C01799=1100.820,324.418,-83.531,179.191,17.633,151.939
C01800=1100.814,324.171,-83.499,179.188,17.631,151.939
C01801=1100.808,323.923,-83.467,179.185,17.628,151.939
C01802=1100.802,323.675,-83.435,179.182,17.626,151.939
C01803=1100.797,323.427,-83.403,179.179,17.624,151.939
C01804=1100.791,323.179,-83.370,179.175,17.622,151.939
C01805=1100.786,322.932,-83.338,179.172,17.619,151.939
C01806=1100.780,322.684,-83.306,179.169,17.617,151.939
C01807=1100.774,322.436,-83.274,179.166,17.614,151.939
C01808=1100.768,322.188,-83.242,179.163,17.612,151.939
C01809=1100.762,321.940,-83.210,179.159,17.609,151.939
C01810=1100.757,321.692,-83.179,179.155,17.607,151.939
C01811=1100.752,321.444,-83.146,179.152,17.604,151.939
C01812=1100.746,321.196,-83.114,179.149,17.602,151.939
C01813=1100.740,320.948,-83.082,179.146,17.599,151.939
C01814=1100.735,320.701,-83.051,179.143,17.597,151.939
C01815=1100.729,320.452,-83.019,179.139,17.595,151.940
C01816=1100.724,320.205,-82.987,179.136,17.593,151.940
C01817=1100.718,319.957,-82.955,179.133,17.590,151.940
C01818=1100.712,319.709,-82.923,179.129,17.588,151.940
C01819=1100.706,319.461,-82.891,179.126,17.586,151.940
C01820=1100.702,319.213,-82.859,179.123,17.583,151.940
C01821=1100.696,318.965,-82.827,179.120,17.581,151.940
C01822=1100.690,318.717,-82.795,179.116,17.579,151.940
C01823=1100.684,318.469,-82.763,179.113,17.576,151.940
C01824=1100.679,318.222,-82.732,179.110,17.574,151.940
C01825=1100.673,317.973,-82.700,179.107,17.572,151.941
C01826=1100.667,317.726,-82.668,179.104,17.569,151.941
C01827=1100.662,317.477,-82.637,179.100,17.566,151.941
C01828=1100.656,317.230,-82.605,179.096,17.564,151.941
C01829=1100.647,316.845,-82.556,179.091,17.561,151.941
C01830=1100.639,316.460,-82.506,179.086,17.558,151.941
C01831=1100.630,316.075,-82.457,179.082,17.554,151.941
C01832=1100.621,315.690,-82.409,179.076,17.550,151.941
C01833=1100.616,315.442,-82.377,179.073,17.548,151.941
C01834=1100.610,315.194,-82.345,179.069,17.546,151.942
C01835=1100.605,314.946,-82.314,179.066,17.543,151.942
C01836=1100.599,314.698,-82.282,179.063,17.541,151.942
C01837=1100.593,314.450,-82.251,179.059,17.539,151.942
C01838=1100.587,314.203,-82.219,179.056,17.537,151.942
C01839=1100.582,313.954,-82.188,179.053,17.535,151.942
C01840=1100.576,313.707,-82.156,179.049,17.533,151.942
C01841=1100.570,313.458,-82.126,179.046,17.531,151.943
C01842=1100.564,313.211,-82.094,179.043,17.529,151.943
C01843=1100.558,312.962,-82.062,179.040,17.527,151.943
C01844=1100.553,312.714,-82.032,179.036,17.525,151.943
C01845=1100.547,312.466,-82.000,179.033,17.523,151.943
C01846=1100.541,312.218,-81.969,179.030,17.520,151.943
C01847=1100.535,311.971,-81.938,179.026,17.518,151.944
C01848=1100.529,311.723,-81.906,179.023,17.516,151.944
C01849=1100.524,311.475,-81.875,179.020,17.514,151.944
C01850=1100.518,311.227,-81.844,179.016,17.512,151.944
C01851=1100.513,310.979,-81.812,179.013,17.510,151.944
C01852=1100.506,310.731,-81.781,179.010,17.508,151.944
C01853=1100.501,310.483,-81.750,179.006,17.506,151.945
C01854=1100.495,310.235,-81.719,179.003,17.504,151.945
C01855=1100.490,309.987,-81.688,178.999,17.502,151.945
C01856=1100.484,309.739,-81.657,178.996,17.499,151.945
C01857=1100.478,309.491,-81.625,178.993,17.497,151.945
C01858=1100.473,309.243,-81.595,178.989,17.495,151.945
C01859=1100.467,308.996,-81.563,178.986,17.493,151.946
C01860=1100.461,308.747,-81.532,178.982,17.491,151.946
C01861=1100.455,308.499,-81.502,178.979,17.489,151.946
C01862=1100.450,308.252,-81.470,178.975,17.487,151.946
C01863=1100.443,308.003,-81.439,178.972,17.485,151.946
C01864=1100.438,307.755,-81.408,178.969,17.483,151.946
C01865=1100.432,307.508,-81.377,178.965,17.481,151.947
C01866=1100.427,307.260,-81.346,178.962,17.479,151.947
C01867=1100.421,307.011,-81.316,178.958,17.477,151.947
C01868=1100.415,306.763,-81.285,178.956,17.476,151.947
C01869=1100.409,306.516,-81.254,178.952,17.474,151.947
C01870=1100.404,306.268,-81.223,178.949,17.472,151.948
C01871=1100.398,306.020,-81.192,178.946,17.470,151.948
C01872=1100.393,305.771,-81.161,178.942,17.467,151.948
C01873=1100.387,305.523,-81.131,178.939,17.465,151.948
C01874=1100.382,305.276,-81.099,178.935,17.463,151.948
C01875=1100.376,305.028,-81.069,178.932,17.461,151.949
C01876=1100.371,304.780,-81.038,178.929,17.459,151.949
C01877=1100.365,304.532,-81.007,178.925,17.457,151.949
C01878=1100.358,304.283,-80.977,178.922,17.455,151.949
C01879=1100.353,304.035,-80.946,178.918,17.453,151.949
C01880=1100.348,303.787,-80.915,178.915,17.451,151.950
C01881=1100.339,303.405,-80.867,178.910,17.448,151.950
C01882=1100.331,303.023,-80.821,178.905,17.445,151.950
C01883=1100.322,302.640,-80.773,178.899,17.442,151.951
C01884=1100.313,302.258,-80.726,178.894,17.439,151.951
C01885=1100.308,302.009,-80.695,178.891,17.437,151.951
C01886=1100.302,301.762,-80.665,178.887,17.435,151.951
C01887=1100.296,301.514,-80.635,178.884,17.433,151.951
C01888=1100.291,301.266,-80.604,178.881,17.432,151.952
C01889=1100.285,301.018,-80.573,178.878,17.430,151.952
C01890=1100.279,300.770,-80.543,178.874,17.428,151.952
C01891=1100.274,300.522,-80.512,178.871,17.426,151.952
C01892=1100.269,300.274,-80.482,178.867,17.424,151.952
C01893=1100.263,300.026,-80.451,178.864,17.422,151.953
C01894=1100.258,299.778,-80.420,178.861,17.420,151.953
C01895=1100.252,299.530,-80.391,178.857,17.418,151.953
C01896=1100.246,299.282,-80.360,178.853,17.416,151.953
C01897=1100.241,299.034,-80.329,178.851,17.415,151.954
C01898=1100.235,298.786,-80.299,178.847,17.413,151.954
C01899=1100.230,298.538,-80.269,178.844,17.411,151.954
C01900=1100.224,298.290,-80.239,178.840,17.409,151.954
C01901=1100.219,298.041,-80.208,178.837,17.407,151.954
C01902=1100.213,297.794,-80.178,178.834,17.405,151.955
C01903=1100.207,297.545,-80.147,178.830,17.403,151.955
C01904=1100.201,297.297,-80.117,178.826,17.401,151.955
C01905=1100.196,297.049,-80.087,178.824,17.400,151.955
C01906=1100.190,296.801,-80.057,178.820,17.398,151.956
C01907=1100.184,296.553,-80.027,178.817,17.396,151.956
C01908=1100.178,296.305,-79.997,178.813,17.394,151.956
C01909=1100.173,296.057,-79.966,178.810,17.392,151.956
C01910=1100.168,295.808,-79.936,178.806,17.390,151.957
C01911=1100.162,295.560,-79.906,178.803,17.389,151.957
C01912=1100.156,295.313,-79.875,178.800,17.387,151.957
C01913=1100.151,295.064,-79.846,178.796,17.385,151.957
C01914=1100.145,294.816,-79.816,178.793,17.384,151.958
C01915=1100.139,294.568,-79.786,178.789,17.382,151.958
C01916=1100.133,294.320,-79.756,178.786,17.380,151.958
C01917=1100.128,294.072,-79.726,178.783,17.379,151.958
C01918=1100.122,293.824,-79.696,178.780,17.377,151.959
C01919=1100.116,293.576,-79.665,178.776,17.375,151.959
C01920=1100.111,293.328,-79.636,178.772,17.373,151.959
C01921=1100.105,293.079,-79.606,178.769,17.371,151.959
C01922=1100.100,292.832,-79.576,178.765,17.369,151.960
C01923=1100.095,292.584,-79.546,178.763,17.368,151.960
C01924=1100.088,292.336,-79.517,178.759,17.366,151.960
C01925=1100.083,292.088,-79.487,178.755,17.364,151.961
C01926=1100.077,291.840,-79.457,178.752,17.362,151.961
C01927=1100.071,291.591,-79.427,178.748,17.361,151.961
C01928=1100.066,291.343,-79.397,178.746,17.359,151.961
C01929=1100.060,291.095,-79.367,178.742,17.357,151.962
C01930=1100.054,290.847,-79.337,178.738,17.356,151.962
C01931=1100.049,290.599,-79.307,178.735,17.354,151.962
C01932=1100.043,290.350,-79.277,178.731,17.352,151.962
C01933=1100.035,289.982,-79.234,178.727,17.350,151.963
C01934=1100.026,289.613,-79.189,178.721,17.347,151.963
C01935=1100.018,289.245,-79.145,178.716,17.345,151.964
C01936=1100.009,288.876,-79.102,178.711,17.343,151.964
C01937=1100.003,288.628,-79.071,178.708,17.341,151.964
C01938=1099.998,288.380,-79.042,178.704,17.339,151.965
C01939=1099.992,288.132,-79.013,178.702,17.338,151.965
C01940=1099.987,287.884,-78.983,178.698,17.336,151.965
C01941=1099.981,287.635,-78.954,178.694,17.334,151.966
C01942=1099.975,287.388,-78.924,178.691,17.333,151.966
C01943=1099.969,287.140,-78.894,178.687,17.331,151.966
C01944=1099.964,286.891,-78.865,178.684,17.330,151.966
C01945=1099.958,286.643,-78.835,178.681,17.328,151.967
C01946=1099.952,286.395,-78.806,178.677,17.326,151.967
C01947=1099.947,286.147,-78.777,178.673,17.325,151.967
C01948=1099.941,285.898,-78.747,178.670,17.324,151.968
C01949=1099.935,285.650,-78.718,178.667,17.322,151.968
C01950=1099.930,285.402,-78.688,178.663,17.320,151.968
C01951=1099.924,285.153,-78.659,178.660,17.318,151.969
C01952=1099.919,284.906,-78.630,178.657,17.317,151.969
C01953=1099.913,284.657,-78.600,178.653,17.316,151.969
C01954=1099.907,284.409,-78.571,178.650,17.314,151.970
C01955=1099.901,284.161,-78.542,178.646,17.312,151.970
C01956=1099.896,283.912,-78.512,178.643,17.311,151.970
C01957=1099.891,283.665,-78.483,178.640,17.309,151.970
C01958=1099.885,283.417,-78.454,178.636,17.308,151.971
C01959=1099.879,283.168,-78.424,178.632,17.306,151.971
C01960=1099.873,282.920,-78.395,178.630,17.305,151.971
C01961=1099.868,282.672,-78.366,178.626,17.303,151.972
C01962=1099.862,282.424,-78.336,178.622,17.301,151.972
C01963=1099.856,282.176,-78.307,178.619,17.300,151.972
C01964=1099.851,281.928,-78.278,178.616,17.298,151.973
C01965=1099.845,281.679,-78.250,178.612,17.297,151.973
C01966=1099.840,281.431,-78.220,178.609,17.295,151.973
C01967=1099.834,281.182,-78.190,178.605,17.293,151.974
C01968=1099.829,280.935,-78.162,178.602,17.292,151.974
C01969=1099.822,280.687,-78.133,178.598,17.291,151.974
C01970=1099.817,280.438,-78.104,178.595,17.289,151.975
C01971=1099.811,280.190,-78.075,178.592,17.288,151.975
C01972=1099.806,279.942,-78.045,178.588,17.286,151.975
C01973=1099.800,279.694,-78.016,178.585,17.284,151.976
C01974=1099.795,279.445,-77.987,178.581,17.283,151.976
C01975=1099.789,279.197,-77.959,178.578,17.282,151.976
C01976=1099.783,278.949,-77.929,178.574,17.280,151.977
C01977=1099.777,278.700,-77.901,178.571,17.278,151.977
C01978=1099.772,278.453,-77.872,178.568,17.277,151.977
C01979=1099.766,278.204,-77.843,178.564,17.276,151.977
C01980=1099.760,277.955,-77.814,178.561,17.274,151.978
C01981=1099.755,277.708,-77.785,178.558,17.273,151.978
C01982=1099.749,277.459,-77.756,178.554,17.271,151.979
C01983=1099.743,277.211,-77.728,178.550,17.270,151.979
C01984=1099.738,276.963,-77.698,178.547,17.268,151.979
C01985=1099.730,276.604,-77.657,178.542,17.266,151.980
C01986=1099.722,276.245,-77.615,178.537,17.264,151.980
C01987=1099.713,275.885,-77.574,178.532,17.262,151.981
C01988=1099.705,275.525,-77.532,178.527,17.260,151.981
C01989=1099.699,275.278,-77.504,178.523,17.258,151.982
C01990=1099.694,275.029,-77.475,178.520,17.257,151.982
C01991=1099.689,274.782,-77.446,178.517,17.256,151.982
C01992=1099.683,274.533,-77.418,178.513,17.254,151.983
C01993=1099.677,274.284,-77.388,178.510,17.253,151.983
C01994=1099.672,274.036,-77.360,178.507,17.251,151.983
C01995=1099.666,273.788,-77.332,178.503,17.250,151.984
C01996=1099.660,273.540,-77.303,178.500,17.249,151.984
C01997=1099.655,273.291,-77.274,178.496,17.247,151.984
C01998=1099.649,273.043,-77.245,178.492,17.246,151.985
C01999=1099.643,272.795,-77.217,178.490,17.245,151.985
C02000=1099.637,272.546,-77.189,178.486,17.243,151.986
C02001=1099.632,272.299,-77.160,178.482,17.241,151.986
C02002=1099.626,272.050,-77.132,178.479,17.240,151.986
C02003=1099.621,271.802,-77.103,178.476,17.239,151.987
C02004=1099.615,271.553,-77.075,178.472,17.237,151.987
C02005=1099.610,271.305,-77.046,178.469,17.236,151.987
C02006=1099.604,271.057,-77.018,178.465,17.235,151.988
C02007=1099.598,270.808,-76.990,178.462,17.233,151.988
C02008=1099.592,270.560,-76.962,178.459,17.232,151.988
C02009=1099.586,270.312,-76.933,178.455,17.231,151.989
C02010=1099.581,270.064,-76.905,178.451,17.229,151.989
C02011=1099.576,269.815,-76.876,178.448,17.228,151.990
C02012=1099.570,269.567,-76.848,178.445,17.227,151.990
C02013=1099.564,269.318,-76.819,178.442,17.226,151.990
C02014=1099.559,269.070,-76.791,178.438,17.224,151.991
C02015=1099.553,268.822,-76.762,178.434,17.223,151.991
C02016=1099.547,268.574,-76.735,178.431,17.222,151.991
C02017=1099.541,268.325,-76.706,178.427,17.220,151.992
C02018=1099.536,268.077,-76.678,178.424,17.219,151.992
C02019=1099.530,267.828,-76.650,178.421,17.218,151.992
C02020=1099.525,267.580,-76.622,178.417,17.216,151.993
C02021=1099.519,267.331,-76.594,178.414,17.215,151.993
C02022=1099.513,267.083,-76.566,178.410,17.214,151.994
C02023=1099.508,266.834,-76.537,178.407,17.212,151.994
C02024=1099.502,266.586,-76.509,178.404,17.211,151.994
C02025=1099.497,266.338,-76.481,178.400,17.210,151.995
C02026=1099.491,266.090,-76.453,178.396,17.208,151.995
C02027=1099.486,265.842,-76.425,178.393,17.207,151.996
C02028=1099.479,265.593,-76.397,178.390,17.206,151.996
C02029=1099.474,265.345,-76.369,178.387,17.205,151.996
C02030=1099.468,265.096,-76.341,178.383,17.203,151.997
C02031=1099.462,264.848,-76.313,178.379,17.202,151.997
C02032=1099.457,264.600,-76.285,178.376,17.201,151.997
C02033=1099.451,264.351,-76.257,178.373,17.199,151.998
C02034=1099.446,264.103,-76.229,178.369,17.198,151.998
C02035=1099.440,263.854,-76.201,178.366,17.197,151.999
C02036=1099.434,263.606,-76.174,178.362,17.196,151.999
C02037=1099.426,263.249,-76.133,178.357,17.194,152.000
C02038=1099.418,262.893,-76.094,178.352,17.192,152.000
C02039=1099.409,262.537,-76.053,178.347,17.190,152.001
C02040=1099.401,262.181,-76.014,178.342,17.189,152.001
C02041=1099.395,261.932,-75.986,178.339,17.188,152.002
C02042=1099.389,261.684,-75.958,178.336,17.187,152.002
C02043=1099.383,261.435,-75.931,178.332,17.185,152.003
C02044=1099.378,261.187,-75.903,178.328,17.184,152.003
C02045=1099.372,260.939,-75.875,178.325,17.183,152.003
C02046=1099.366,260.690,-75.847,178.321,17.182,152.004
C02047=1099.361,260.442,-75.820,178.318,17.181,152.004
C02048=1099.355,260.194,-75.792,178.315,17.179,152.005
C02049=1099.349,259.945,-75.764,178.311,17.178,152.005
C02050=1099.344,259.696,-75.737,178.308,17.177,152.006
C02051=1099.337,259.448,-75.709,178.304,17.175,152.006
C02052=1099.332,259.200,-75.681,178.301,17.175,152.006
C02053=1099.327,258.951,-75.654,178.297,17.173,152.007
C02054=1099.320,258.703,-75.626,178.294,17.172,152.007
C02055=1099.315,258.454,-75.599,178.290,17.171,152.008
C02056=1099.310,258.206,-75.571,178.287,17.170,152.008
C02057=1099.304,257.958,-75.544,178.284,17.169,152.008
C02058=1099.298,257.709,-75.516,178.280,17.167,152.009
C02059=1099.292,257.461,-75.489,178.277,17.166,152.009
C02060=1099.287,257.213,-75.461,178.273,17.165,152.010
C02061=1099.281,256.963,-75.434,178.270,17.164,152.010
C02062=1099.275,256.715,-75.406,178.266,17.162,152.010
C02063=1099.270,256.467,-75.379,178.263,17.162,152.011
C02064=1099.264,256.219,-75.352,178.259,17.160,152.011
C02065=1099.259,255.970,-75.324,178.256,17.159,152.012
C02066=1099.252,255.722,-75.297,178.253,17.158,152.012
C02067=1099.247,255.473,-75.270,178.249,17.156,152.012
C02068=1099.242,255.225,-75.242,178.246,17.156,152.013
C02069=1099.236,254.976,-75.215,178.242,17.154,152.013
C02070=1099.231,254.727,-75.187,178.239,17.154,152.014
C02071=1099.225,254.480,-75.160,178.235,17.152,152.014
C02072=1099.220,254.231,-75.133,178.232,17.151,152.015
C02073=1099.213,253.982,-75.106,178.228,17.150,152.015
C02074=1099.208,253.734,-75.078,178.225,17.149,152.015
C02075=1099.202,253.486,-75.051,178.222,17.147,152.016
C02076=1099.197,253.237,-75.024,178.218,17.146,152.016
C02077=1099.191,252.989,-74.997,178.215,17.145,152.017
C02078=1099.186,252.741,-74.969,178.211,17.144,152.017
C02079=1099.180,252.491,-74.942,178.208,17.143,152.018
C02080=1099.175,252.243,-74.915,178.204,17.141,152.018
C02081=1099.169,251.994,-74.888,178.201,17.141,152.018
C02082=1099.163,251.746,-74.860,178.198,17.139,152.019
C02083=1099.158,251.498,-74.834,178.194,17.139,152.019
C02084=1099.152,251.250,-74.807,178.191,17.137,152.020
C02085=1099.146,251.000,-74.780,178.188,17.136,152.020
C02086=1099.140,250.752,-74.753,178.184,17.135,152.020
C02087=1099.135,250.504,-74.725,178.181,17.134,152.021
C02088=1099.129,250.256,-74.698,178.177,17.133,152.021
C02089=1099.121,249.896,-74.659,178.172,17.131,152.022
C02090=1099.113,249.537,-74.620,178.167,17.129,152.022
C02091=1099.105,249.178,-74.581,178.162,17.127,152.023
C02092=1099.098,248.818,-74.543,178.157,17.126,152.024
C02093=1099.093,248.569,-74.516,178.154,17.125,152.024
C02094=1099.087,248.321,-74.489,178.151,17.124,152.024
C02095=1099.081,248.073,-74.462,178.147,17.122,152.025
C02096=1099.076,247.824,-74.435,178.144,17.122,152.025
C02097=1099.070,247.576,-74.408,178.140,17.120,152.026
C02098=1099.064,247.327,-74.381,178.137,17.119,152.026
C02099=1099.059,247.078,-74.354,178.133,17.118,152.027
C02100=1099.053,246.830,-74.328,178.130,17.117,152.027
C02101=1099.047,246.581,-74.301,178.126,17.116,152.027
C02102=1099.042,246.333,-74.274,178.123,17.115,152.028
C02103=1099.037,246.084,-74.247,178.119,17.114,152.028
C02104=1099.031,245.836,-74.220,178.116,17.113,152.029
C02105=1099.025,245.587,-74.194,178.113,17.111,152.029
C02106=1099.019,245.339,-74.167,178.110,17.111,152.030
C02107=1099.013,245.091,-74.140,178.106,17.109,152.030
C02108=1099.009,244.841,-74.114,178.103,17.108,152.030
C02109=1099.003,244.593,-74.087,178.099,17.107,152.031
C02110=1098.997,244.345,-74.061,178.096,17.106,152.031
C02111=1098.991,244.096,-74.034,178.092,17.105,152.032
C02112=1098.986,243.848,-74.007,178.089,17.104,152.032
C02113=1098.980,243.600,-73.981,178.085,17.103,152.033
C02114=1098.975,243.350,-73.954,178.082,17.102,152.033
C02115=1098.969,243.102,-73.927,178.078,17.101,152.034
C02116=1098.964,242.854,-73.901,178.075,17.100,152.034
C02117=1098.958,242.605,-73.874,178.072,17.099,152.034
C02118=1098.952,242.356,-73.848,178.068,17.098,152.035
C02119=1098.947,242.108,-73.822,178.065,17.097,152.035
C02120=1098.941,241.860,-73.795,178.061,17.096,152.036
C02121=1098.935,241.611,-73.769,178.058,17.095,152.036
C02122=1098.930,241.362,-73.742,178.054,17.094,152.037
C02123=1098.924,241.114,-73.716,178.051,17.093,152.037
C02124=1098.918,240.865,-73.690,178.048,17.092,152.038
C02125=1098.913,240.617,-73.663,178.044,17.091,152.038
C02126=1098.907,240.368,-73.636,178.041,17.090,152.039
C02127=1098.901,240.119,-73.611,178.037,17.089,152.039
C02128=1098.896,239.871,-73.584,178.034,17.088,152.039
C02129=1098.890,239.622,-73.558,178.030,17.087,152.040
C02130=1098.884,239.374,-73.531,178.028,17.086,152.040
C02131=1098.879,239.125,-73.505,178.024,17.085,152.041
C02132=1098.873,238.876,-73.479,178.021,17.084,152.041
C02133=1098.867,238.628,-73.452,178.017,17.083,152.042
C02134=1098.861,238.379,-73.427,178.014,17.082,152.042
C02135=1098.856,238.132,-73.400,178.010,17.081,152.043
C02136=1098.850,237.883,-73.375,178.007,17.080,152.043
C02137=1098.845,237.634,-73.348,178.004,17.079,152.044
C02138=1098.839,237.385,-73.322,178.000,17.078,152.044
C02139=1098.833,237.137,-73.295,177.997,17.077,152.044
C02140=1098.828,236.888,-73.269,177.993,17.076,152.045
C02141=1098.819,236.521,-73.231,177.988,17.075,152.046
C02142=1098.812,236.156,-73.192,177.983,17.073,152.046
C02143=1098.803,235.789,-73.154,177.978,17.072,152.047
C02144=1098.794,235.423,-73.116,177.973,17.070,152.048
C02145=1098.790,235.175,-73.090,177.970,17.070,152.048
C02146=1098.784,234.926,-73.064,177.966,17.068,152.048
C02147=1098.778,234.677,-73.038,177.963,17.068,152.049
C02148=1098.773,234.428,-73.012,177.959,17.066,152.049
C02149=1098.766,234.180,-72.986,177.956,17.066,152.050
C02150=1098.761,233.932,-72.960,177.953,17.065,152.050
C02151=1098.756,233.683,-72.934,177.949,17.064,152.051
C02152=1098.750,233.434,-72.908,177.946,17.063,152.051
C02153=1098.745,233.186,-72.882,177.942,17.062,152.052
C02154=1098.739,232.937,-72.856,177.939,17.061,152.052
C02155=1098.733,232.688,-72.830,177.936,17.060,152.053
C02156=1098.728,232.440,-72.805,177.932,17.059,152.053
C02157=1098.722,232.192,-72.779,177.929,17.058,152.054
C02158=1098.716,231.943,-72.753,177.925,17.057,152.054
C02159=1098.711,231.694,-72.727,177.922,17.056,152.054
C02160=1098.705,231.445,-72.701,177.919,17.055,152.055
C02161=1098.700,231.197,-72.676,177.915,17.054,152.055
C02162=1098.694,230.948,-72.650,177.912,17.053,152.056
C02163=1098.688,230.700,-72.623,177.908,17.052,152.056
C02164=1098.682,230.451,-72.598,177.905,17.052,152.057
C02165=1098.677,230.203,-72.572,177.902,17.051,152.057
C02166=1098.671,229.954,-72.547,177.898,17.050,152.058
C02167=1098.666,229.705,-72.521,177.895,17.049,152.058
C02168=1098.660,229.456,-72.495,177.891,17.048,152.059
C02169=1098.655,229.208,-72.470,177.888,17.047,152.059
C02170=1098.649,228.959,-72.444,177.885,17.046,152.060
C02171=1098.643,228.710,-72.419,177.881,17.045,152.060
C02172=1098.637,228.461,-72.393,177.878,17.044,152.061
C02173=1098.632,228.213,-72.368,177.875,17.043,152.061
C02174=1098.626,227.964,-72.342,177.871,17.042,152.062
C02175=1098.620,227.716,-72.317,177.868,17.042,152.062
C02176=1098.615,227.467,-72.291,177.864,17.040,152.063
C02177=1098.609,227.219,-72.266,177.861,17.040,152.063
C02178=1098.604,226.970,-72.240,177.858,17.039,152.063
C02179=1098.597,226.721,-72.215,177.854,17.038,152.064
C02180=1098.593,226.473,-72.189,177.851,17.037,152.064
C02181=1098.586,226.224,-72.164,177.847,17.037,152.065
C02182=1098.581,225.975,-72.138,177.844,17.035,152.065
C02183=1098.576,225.727,-72.114,177.840,17.035,152.066
C02184=1098.570,225.478,-72.088,177.838,17.034,152.066
C02185=1098.564,225.229,-72.062,177.834,17.033,152.067
C02186=1098.559,224.981,-72.037,177.831,17.032,152.067
C02187=1098.553,224.732,-72.011,177.827,17.031,152.068
C02188=1098.547,224.483,-71.985,177.824,17.030,152.068
C02189=1098.542,224.234,-71.961,177.820,17.029,152.069
C02190=1098.536,223.986,-71.936,177.817,17.028,152.069
C02191=1098.530,223.737,-71.910,177.813,17.027,152.070
C02192=1098.525,223.489,-71.885,177.810,17.026,152.070
C02193=1098.517,223.113,-71.847,177.805,17.025,152.071
C02194=1098.509,222.739,-71.809,177.800,17.024,152.072
C02195=1098.499,222.365,-71.771,177.795,17.023,152.072
C02196=1098.491,221.989,-71.733,177.790,17.021,152.073
C02197=1098.486,221.741,-71.708,177.786,17.020,152.073
C02198=1098.480,221.492,-71.682,177.783,17.020,152.074
C02199=1098.474,221.243,-71.658,177.780,17.019,152.074
C02200=1098.469,220.995,-71.633,177.776,17.018,152.075
C02201=1098.463,220.747,-71.607,177.773,17.017,152.075
C02202=1098.458,220.498,-71.582,177.770,17.016,152.076
C02203=1098.452,220.249,-71.557,177.766,17.015,152.076
C02204=1098.446,220.000,-71.533,177.763,17.014,152.077
C02205=1098.440,219.752,-71.508,177.760,17.014,152.077
C02206=1098.434,219.503,-71.482,177.756,17.013,152.078
C02207=1098.429,219.254,-71.457,177.753,17.012,152.078
C02208=1098.423,219.005,-71.432,177.749,17.012,152.079
C02209=1098.418,218.757,-71.408,177.746,17.010,152.079
C02210=1098.412,218.508,-71.382,177.742,17.010,152.080
C02211=1098.406,218.260,-71.358,177.739,17.009,152.080
C02212=1098.401,218.011,-71.332,177.735,17.008,152.081
C02213=1098.395,217.761,-71.308,177.732,17.007,152.081
C02214=1098.390,217.513,-71.283,177.729,17.006,152.082
C02215=1098.384,217.264,-71.258,177.726,17.006,152.082
C02216=1098.378,217.016,-71.233,177.722,17.005,152.083
C02217=1098.373,216.766,-71.208,177.719,17.004,152.083
C02218=1098.368,216.518,-71.184,177.716,17.003,152.084
C02219=1098.362,216.270,-71.159,177.712,17.002,152.084
C02220=1098.356,216.021,-71.134,177.709,17.001,152.085
C02221=1098.350,215.773,-71.109,177.706,17.001,152.085
C02222=1098.345,215.523,-71.084,177.702,17.000,152.086
C02223=1098.339,215.275,-71.060,177.699,16.999,152.086
C02224=1098.333,215.026,-71.035,177.696,16.998,152.087
C02225=1098.328,214.777,-71.010,177.693,16.998,152.087
C02226=1098.323,214.528,-70.985,177.689,16.996,152.088
C02227=1098.317,214.280,-70.960,177.686,16.996,152.088
C02228=1098.311,214.031,-70.936,177.682,16.995,152.088
C02229=1098.306,213.782,-70.911,177.679,16.994,152.089
C02230=1098.300,213.534,-70.887,177.675,16.993,152.089
C02231=1098.294,213.285,-70.862,177.672,16.993,152.090
C02232=1098.289,213.036,-70.838,177.669,16.992,152.090
C02233=1098.283,212.787,-70.813,177.665,16.991,152.091
C02234=1098.278,212.538,-70.789,177.662,16.990,152.091
C02235=1098.272,212.290,-70.764,177.659,16.990,152.092
C02236=1098.266,212.041,-70.739,177.655,16.988,152.092
C02237=1098.261,211.793,-70.715,177.652,16.988,152.093
C02238=1098.255,211.543,-70.690,177.649,16.987,152.093
C02239=1098.250,211.295,-70.666,177.646,16.986,152.094
C02240=1098.244,211.047,-70.641,177.642,16.985,152.094
C02241=1098.238,210.797,-70.616,177.639,16.985,152.095
C02242=1098.233,210.549,-70.592,177.636,16.984,152.095
C02243=1098.227,210.300,-70.568,177.632,16.983,152.096
C02244=1098.221,210.051,-70.544,177.629,16.982,152.096
C02245=1098.213,209.681,-70.507,177.623,16.981,152.097
C02246=1098.205,209.309,-70.470,177.619,16.980,152.098
C02247=1098.196,208.939,-70.434,177.614,16.979,152.099
C02248=1098.188,208.568,-70.399,177.609,16.978,152.099
C02249=1098.165,207.558,-70.300,177.564,16.962,152.105
C02250=1098.159,207.309,-70.276,177.560,16.962,152.105
C02251=1098.154,207.060,-70.253,177.557,16.962,152.106
C02252=1098.148,206.811,-70.228,177.553,16.962,152.107
C02253=1098.142,206.562,-70.204,177.550,16.962,152.108
C02254=1098.137,206.314,-70.180,177.546,16.962,152.108
C02255=1098.131,206.065,-70.156,177.543,16.962,152.109
C02256=1098.125,205.816,-70.133,177.539,16.962,152.110
C02257=1098.120,205.567,-70.108,177.536,16.962,152.110
C02258=1098.114,205.319,-70.084,177.532,16.962,152.111
C02259=1098.108,205.070,-70.060,177.529,16.962,152.112
C02260=1098.103,204.820,-70.037,177.525,16.962,152.113
C02261=1098.097,204.572,-70.012,177.522,16.963,152.113
C02262=1098.091,204.323,-69.989,177.519,16.963,152.114
C02263=1098.086,204.075,-69.964,177.515,16.963,152.115
C02264=1098.081,203.826,-69.941,177.512,16.963,152.115
C02265=1098.075,203.577,-69.917,177.508,16.963,152.116
C02266=1098.069,203.328,-69.893,177.505,16.963,152.117
C02267=1098.063,203.079,-69.870,177.501,16.963,152.117
C02268=1098.058,202.831,-69.845,177.498,16.963,152.118
C02269=1098.052,202.582,-69.822,177.494,16.964,152.119
C02270=1098.047,202.333,-69.798,177.490,16.964,152.120
C02271=1098.041,202.084,-69.774,177.487,16.964,152.120
C02272=1098.036,201.835,-69.751,177.483,16.964,152.121
C02273=1098.029,201.587,-69.727,177.480,16.964,152.122
C02274=1098.024,201.338,-69.703,177.476,16.964,152.123
C02275=1098.018,201.088,-69.679,177.473,16.964,152.123
C02276=1098.012,200.840,-69.656,177.469,16.964,152.124
C02277=1098.007,200.591,-69.632,177.466,16.964,152.125
C02278=1098.001,200.343,-69.608,177.463,16.965,152.125
C02279=1097.996,200.094,-69.585,177.459,16.965,152.126
C02280=1097.990,199.845,-69.561,177.456,16.965,152.127
C02281=1097.983,199.596,-69.538,177.452,16.965,152.128
C02282=1097.978,199.347,-69.514,177.449,16.965,152.128
C02283=1097.972,199.098,-69.491,177.445,16.965,152.129
C02284=1097.967,198.850,-69.467,177.442,16.965,152.130
C02285=1097.961,198.601,-69.444,177.438,16.965,152.130
C02286=1097.955,198.352,-69.420,177.435,16.965,152.131
C02287=1097.950,198.103,-69.396,177.431,16.965,152.132
C02288=1097.944,197.854,-69.372,177.427,16.965,152.132
C02289=1097.938,197.605,-69.349,177.424,16.965,152.133
C02290=1097.933,197.356,-69.326,177.420,16.965,152.134
C02291=1097.927,197.108,-69.302,177.418,16.966,152.135
C02292=1097.921,196.859,-69.279,177.414,16.966,152.135
C02293=1097.916,196.610,-69.255,177.411,16.966,152.136
C02294=1097.910,196.361,-69.232,177.407,16.966,152.137
C02295=1097.904,196.113,-69.209,177.404,16.966,152.137
C02296=1097.899,195.864,-69.185,177.400,16.966,152.138
C02297=1097.893,195.615,-69.162,177.396,16.966,152.139
C02298=1097.888,195.366,-69.139,177.393,16.966,152.140
C02299=1097.882,195.117,-69.114,177.389,16.966,152.140
C02300=1097.876,194.868,-69.091,177.386,16.966,152.141
C02301=1097.870,194.619,-69.068,177.383,16.966,152.142
C02302=1097.865,194.370,-69.045,177.379,16.966,152.142
C02303=1097.859,194.122,-69.021,177.376,16.966,152.143
C02304=1097.854,193.873,-68.998,177.373,16.966,152.144
C02305=1097.848,193.624,-68.975,177.369,16.966,152.144
C02306=1097.842,193.375,-68.952,177.366,16.966,152.145
C02307=1097.837,193.126,-68.929,177.362,16.967,152.146
C02308=1097.831,192.877,-68.905,177.359,16.966,152.146
C02309=1097.825,192.629,-68.882,177.355,16.966,152.147
C02310=1097.819,192.354,-68.857,177.352,16.966,152.148
C02311=1097.813,192.080,-68.832,177.348,16.967,152.149
C02312=1097.807,191.807,-68.805,177.345,16.967,152.149
C02313=1097.801,191.533,-68.780,177.340,16.966,152.150
C02314=1097.795,191.284,-68.757,177.337,16.966,152.151
C02315=1097.790,191.035,-68.734,177.334,16.967,152.151
C02316=1097.784,190.786,-68.711,177.331,16.967,152.152
C02317=1097.779,190.537,-68.688,177.327,16.967,152.153
C02318=1097.773,190.288,-68.665,177.324,16.967,152.153
C02319=1097.768,190.039,-68.642,177.320,16.967,152.154
C02320=1097.762,189.790,-68.619,177.317,16.966,152.155
C02321=1097.757,189.542,-68.596,177.313,16.966,152.155
C02322=1097.752,189.293,-68.573,177.310,16.966,152.156
C02323=1097.746,189.044,-68.550,177.306,16.966,152.157
C02324=1097.740,188.795,-68.527,177.303,16.966,152.157
C02325=1097.734,188.546,-68.504,177.300,16.967,152.158
C02326=1097.729,188.297,-68.481,177.297,16.967,152.159
C02327=1097.723,188.048,-68.458,177.293,16.966,152.159
C02328=1097.718,187.799,-68.434,177.290,16.966,152.160
C02329=1097.712,187.550,-68.411,177.286,16.966,152.161
C02330=1097.707,187.302,-68.389,177.283,16.966,152.161
C02331=1097.701,187.053,-68.366,177.280,16.966,152.162
C02332=1097.696,186.804,-68.343,177.276,16.966,152.163
C02333=1097.690,186.555,-68.320,177.274,16.966,152.163
C02334=1097.684,186.306,-68.297,177.270,16.966,152.164
C02335=1097.678,186.057,-68.274,177.267,16.966,152.165
C02336=1097.674,185.809,-68.251,177.263,16.966,152.165
C02337=1097.669,185.559,-68.229,177.260,16.966,152.166
C02338=1097.663,185.310,-68.206,177.257,16.966,152.167
C02339=1097.657,185.062,-68.183,177.253,16.966,152.167
C02340=1097.651,184.813,-68.160,177.249,16.966,152.168
C02341=1097.645,184.564,-68.137,177.247,16.967,152.169
C02342=1097.639,184.315,-68.115,177.243,16.966,152.169
C02343=1097.634,184.066,-68.092,177.240,16.966,152.170
C02344=1097.628,183.817,-68.069,177.236,16.966,152.171
C02345=1097.622,183.568,-68.046,177.233,16.966,152.171
C02346=1097.617,183.320,-68.024,177.230,16.966,152.172
C02347=1097.611,183.071,-68.001,177.226,16.966,152.173
C02348=1097.605,182.822,-67.979,177.223,16.967,152.173
C02349=1097.600,182.573,-67.956,177.220,16.967,152.174
C02350=1097.594,182.324,-67.933,177.217,16.966,152.175
C02351=1097.588,182.075,-67.912,177.213,16.966,152.175
C02352=1097.582,181.826,-67.889,177.209,16.966,152.176
C02353=1097.576,181.577,-67.866,177.206,16.966,152.177
C02354=1097.571,181.329,-67.843,177.203,16.966,152.177
C02355=1097.565,181.079,-67.822,177.200,16.967,152.178
C02356=1097.559,180.831,-67.799,177.196,16.967,152.179
C02357=1097.554,180.582,-67.776,177.193,16.966,152.179
C02358=1097.548,180.332,-67.753,177.190,16.967,152.180
C02359=1097.542,180.084,-67.731,177.186,16.967,152.181
C02360=1097.537,179.835,-67.709,177.183,16.966,152.181
C02361=1097.531,179.586,-67.686,177.179,16.966,152.182
C02362=1097.525,179.337,-67.663,177.177,16.967,152.183
C02363=1097.519,179.088,-67.642,177.173,16.967,152.183
C02364=1097.513,178.839,-67.619,177.170,16.967,152.184
C02365=1097.509,178.590,-67.597,177.167,16.966,152.185
C02366=1097.502,178.341,-67.575,177.163,16.966,152.185
C02367=1097.497,178.092,-67.552,177.160,16.966,152.186
C02368=1097.491,177.843,-67.529,177.157,16.967,152.187
C02369=1097.485,177.594,-67.508,177.153,16.967,152.187
C02370=1097.480,177.346,-67.485,177.150,16.966,152.188
C02371=1097.474,177.096,-67.463,177.147,16.966,152.189
C02372=1097.468,176.847,-67.441,177.143,16.966,152.189
C02373=1097.462,176.598,-67.418,177.140,16.966,152.190
C02374=1097.456,176.324,-67.393,177.136,16.966,152.191
C02375=1097.450,176.050,-67.369,177.133,16.966,152.191
C02376=1097.444,175.775,-67.345,177.130,16.966,152.192
C02377=1097.438,175.501,-67.319,177.126,16.966,152.193
C02378=1097.432,175.252,-67.298,177.122,16.966,152.193
C02379=1097.427,175.003,-67.276,177.119,16.966,152.194
C02380=1097.420,174.754,-67.254,177.116,16.966,152.195
C02381=1097.415,174.505,-67.232,177.113,16.966,152.195
C02382=1097.410,174.257,-67.209,177.110,16.966,152.196
C02383=1097.403,174.007,-67.187,177.106,16.966,152.196
C02384=1097.399,173.759,-67.165,177.103,16.966,152.197
C02385=1097.392,173.510,-67.143,177.100,16.965,152.198
C02386=1097.387,173.260,-67.121,177.096,16.965,152.198
C02387=1097.382,173.012,-67.099,177.094,16.966,152.199
C02388=1097.375,172.763,-67.076,177.090,16.965,152.199
C02389=1097.370,172.513,-67.054,177.087,16.965,152.200
C02390=1097.364,172.265,-67.033,177.084,16.965,152.201
C02391=1097.359,172.015,-67.011,177.080,16.965,152.201
C02392=1097.353,171.767,-66.988,177.078,16.965,152.202
C02393=1097.348,171.518,-66.966,177.074,16.965,152.203
C02394=1097.342,171.269,-66.944,177.071,16.964,152.203
C02395=1097.337,171.020,-66.923,177.068,16.965,152.204
C02396=1097.331,170.771,-66.900,177.064,16.964,152.204
C02397=1097.325,170.522,-66.878,177.061,16.964,152.205
C02398=1097.320,170.273,-66.857,177.058,16.964,152.206
C02399=1097.314,170.024,-66.835,177.055,16.964,152.206
C02400=1097.309,169.775,-66.813,177.052,16.964,152.207
C02401=1097.304,169.526,-66.791,177.048,16.964,152.208
C02402=1097.298,169.278,-66.769,177.045,16.963,152.208
C02403=1097.292,169.028,-66.747,177.043,16.964,152.209
C02404=1097.286,168.779,-66.725,177.039,16.964,152.209
C02405=1097.281,168.530,-66.703,177.036,16.963,152.210
C02406=1097.275,168.281,-66.681,177.033,16.963,152.210
C02407=1097.270,168.032,-66.660,177.029,16.963,152.211
C02408=1097.264,167.783,-66.638,177.027,16.963,152.212
C02409=1097.259,167.534,-66.616,177.023,16.963,152.212
C02410=1097.253,167.285,-66.594,177.020,16.963,152.213
C02411=1097.248,167.036,-66.573,177.017,16.962,152.213
C02412=1097.242,166.787,-66.551,177.013,16.962,152.214
C02413=1097.237,166.538,-66.529,177.011,16.962,152.215
C02414=1097.231,166.289,-66.507,177.008,16.962,152.215
C02415=1097.226,166.040,-66.486,177.004,16.962,152.216
C02416=1097.220,165.791,-66.464,177.001,16.961,152.216
C02417=1097.215,165.542,-66.443,176.998,16.961,152.217
C02418=1097.209,165.293,-66.420,176.995,16.962,152.218
C02419=1097.204,165.044,-66.399,176.992,16.961,152.218
C02420=1097.198,164.795,-66.377,176.988,16.961,152.219
C02421=1097.193,164.546,-66.356,176.985,16.961,152.219
C02422=1097.187,164.297,-66.333,176.982,16.960,152.220
C02423=1097.182,164.048,-66.312,176.980,16.960,152.220
C02424=1097.176,163.799,-66.291,176.976,16.960,152.221
C02425=1097.171,163.550,-66.269,176.973,16.960,152.222
C02426=1097.165,163.302,-66.247,176.969,16.960,152.222
C02427=1097.160,163.052,-66.225,176.966,16.959,152.223
C02428=1097.155,162.803,-66.205,176.964,16.960,152.223
C02429=1097.148,162.554,-66.183,176.961,16.959,152.224
C02430=1097.144,162.305,-66.161,176.957,16.959,152.225
C02431=1097.138,162.057,-66.140,176.954,16.959,152.225
C02432=1097.133,161.807,-66.118,176.951,16.958,152.226
C02433=1097.127,161.559,-66.096,176.948,16.958,152.226
C02434=1097.121,161.309,-66.075,176.945,16.958,152.227
C02435=1097.116,161.060,-66.054,176.942,16.958,152.227
C02436=1097.109,160.811,-66.033,176.938,16.958,152.228
C02437=1097.105,160.562,-66.011,176.935,16.957,152.229
C02438=1097.098,160.287,-65.987,176.932,16.957,152.229
C02439=1097.092,160.013,-65.964,176.928,16.957,152.230
C02440=1097.085,159.738,-65.940,176.925,16.957,152.230
C02441=1097.079,159.463,-65.917,176.922,16.956,152.231
C02442=1097.074,159.214,-65.896,176.918,16.957,152.232
C02443=1097.067,158.965,-65.874,176.916,16.957,152.232
C02444=1097.063,158.716,-65.853,176.912,16.956,152.233
C02445=1097.057,158.467,-65.832,176.909,16.956,152.233
C02446=1097.051,158.218,-65.810,176.906,16.956,152.234
C02447=1097.046,157.970,-65.789,176.903,16.956,152.235
C02448=1097.040,157.720,-65.768,176.900,16.956,152.235
C02449=1097.034,157.471,-65.747,176.897,16.955,152.236
C02450=1097.029,157.222,-65.726,176.894,16.955,152.236
C02451=1097.023,156.973,-65.704,176.891,16.955,152.237
C02452=1097.018,156.724,-65.683,176.888,16.955,152.237
C02453=1097.013,156.475,-65.662,176.885,16.954,152.238
C02454=1097.007,156.226,-65.640,176.881,16.954,152.239
C02455=1097.001,155.977,-65.620,176.879,16.954,152.239
C02456=1096.995,155.727,-65.598,176.876,16.954,152.240
C02457=1096.990,155.479,-65.577,176.872,16.953,152.240
C02458=1096.984,155.230,-65.556,176.869,16.953,152.241
C02459=1096.978,154.981,-65.535,176.866,16.953,152.241
C02460=1096.973,154.731,-65.514,176.863,16.953,152.242
C02461=1096.967,154.483,-65.493,176.860,16.953,152.242
C02462=1096.961,154.233,-65.472,176.857,16.952,152.243
C02463=1096.956,153.985,-65.451,176.854,16.952,152.244
C02464=1096.951,153.736,-65.430,176.851,16.952,152.244
C02465=1096.945,153.486,-65.409,176.848,16.952,152.245
C02466=1096.939,153.237,-65.388,176.845,16.951,152.245
C02467=1096.934,152.989,-65.367,176.841,16.951,152.246
C02468=1096.928,152.739,-65.346,176.839,16.951,152.246
C02469=1096.922,152.490,-65.325,176.836,16.951,152.247
C02470=1096.917,152.241,-65.304,176.832,16.951,152.247
C02471=1096.911,151.991,-65.283,176.829,16.950,152.248
C02472=1096.905,151.743,-65.262,176.827,16.951,152.249
C02473=1096.900,151.494,-65.242,176.824,16.950,152.249
C02474=1096.893,151.245,-65.220,176.821,16.949,152.250
C02475=1096.888,150.996,-65.200,176.817,16.949,152.250
C02476=1096.883,150.747,-65.179,176.815,16.949,152.251
C02477=1096.877,150.498,-65.158,176.812,16.949,152.251
C02478=1096.872,150.248,-65.137,176.808,16.949,152.252
C02479=1096.866,149.999,-65.116,176.806,16.949,152.252
C02480=1096.861,149.751,-65.095,176.803,16.948,152.253
C02481=1096.855,149.502,-65.075,176.800,16.948,152.253
C02482=1096.849,149.252,-65.054,176.796,16.947,152.254
C02483=1096.843,149.004,-65.033,176.794,16.947,152.254
C02484=1096.838,148.754,-65.012,176.791,16.947,152.255
C02485=1096.833,148.505,-64.992,176.787,16.947,152.256
C02486=1096.827,148.255,-64.971,176.784,16.946,152.256
C02487=1096.821,148.007,-64.950,176.782,16.946,152.257
C02488=1096.815,147.758,-64.930,176.779,16.946,152.257
C02489=1096.810,147.509,-64.909,176.775,16.945,152.258
C02490=1096.804,147.259,-64.888,176.772,16.945,152.258
C02491=1096.799,147.011,-64.867,176.770,16.945,152.259
C02492=1096.793,146.762,-64.847,176.767,16.945,152.259
C02493=1096.787,146.513,-64.826,176.763,16.944,152.260
C02494=1096.782,146.263,-64.806,176.761,16.944,152.260
C02495=1096.776,146.014,-64.786,176.758,16.944,152.261
C02496=1096.770,145.765,-64.765,176.754,16.944,152.262
C02497=1096.765,145.516,-64.744,176.752,16.943,152.262
C02498=1096.760,145.267,-64.723,176.749,16.943,152.262
C02499=1096.753,145.018,-64.703,176.746,16.943,152.263
C02500=1096.748,144.769,-64.682,176.743,16.942,152.264
C02501=1096.742,144.520,-64.662,176.740,16.942,152.264
C02502=1096.735,144.245,-64.639,176.736,16.941,152.265
C02503=1096.730,143.970,-64.617,176.733,16.941,152.265
C02504=1096.724,143.695,-64.594,176.730,16.941,152.266
C02505=1096.717,143.420,-64.572,176.727,16.940,152.266
C02506=1096.712,143.171,-64.551,176.724,16.941,152.267
C02507=1096.707,142.922,-64.531,176.721,16.940,152.267
C02508=1096.701,142.673,-64.511,176.718,16.939,152.268
C02509=1096.695,142.424,-64.489,176.715,16.940,152.268
C02510=1096.689,142.174,-64.469,176.712,16.939,152.269
C02511=1096.683,141.926,-64.449,176.709,16.938,152.269
C02512=1096.678,141.676,-64.428,176.706,16.938,152.270
C02513=1096.673,141.427,-64.408,176.704,16.938,152.270
C02514=1096.667,141.178,-64.388,176.700,16.938,152.271
C02515=1096.662,140.929,-64.368,176.697,16.937,152.271
C02516=1096.656,140.680,-64.347,176.695,16.937,152.272
C02517=1096.650,140.431,-64.327,176.692,16.937,152.272
C02518=1096.645,140.181,-64.306,176.688,16.936,152.273
C02519=1096.639,139.932,-64.286,176.686,16.936,152.273
C02520=1096.633,139.683,-64.266,176.683,16.936,152.274
C02521=1096.627,139.434,-64.246,176.680,16.935,152.274
C02522=1096.622,139.185,-64.225,176.677,16.935,152.275
C02523=1096.616,138.936,-64.205,176.674,16.935,152.276
C02524=1096.611,138.687,-64.185,176.671,16.934,152.276
C02525=1096.605,138.438,-64.165,176.668,16.934,152.277
C02526=1096.600,138.189,-64.145,176.666,16.933,152.277
C02527=1096.594,137.940,-64.125,176.663,16.933,152.277
C02528=1096.588,137.690,-64.104,176.660,16.932,152.278
C02529=1096.582,137.441,-64.084,176.657,16.933,152.278
C02530=1096.577,137.192,-64.064,176.654,16.932,152.279
C02531=1096.571,136.943,-64.044,176.651,16.931,152.279
C02532=1096.566,136.693,-64.024,176.648,16.931,152.280
C02533=1096.560,136.445,-64.004,176.646,16.931,152.280
C02534=1096.555,136.196,-63.983,176.642,16.931,152.281
C02535=1096.549,135.947,-63.963,176.639,16.930,152.281
C02536=1096.543,135.697,-63.944,176.637,16.930,152.282
C02537=1096.538,135.448,-63.923,176.634,16.929,152.282
C02538=1096.532,135.199,-63.904,176.631,16.929,152.283
C02539=1096.526,134.950,-63.883,176.628,16.929,152.283
C02540=1096.521,134.701,-63.864,176.625,16.928,152.284
C02541=1096.515,134.452,-63.844,176.622,16.928,152.284
C02542=1096.509,134.203,-63.823,176.620,16.928,152.285
C02543=1096.504,133.953,-63.804,176.617,16.927,152.285
C02544=1096.498,133.704,-63.783,176.613,16.927,152.286
C02545=1096.492,133.456,-63.763,176.611,16.926,152.286
C02546=1096.487,133.206,-63.744,176.608,16.926,152.287
C02547=1096.482,132.957,-63.724,176.605,16.925,152.287
C02548=1096.476,132.708,-63.704,176.602,16.924,152.288
C02549=1096.471,132.458,-63.684,176.600,16.925,152.288
C02550=1096.465,132.210,-63.664,176.597,16.924,152.289
C02551=1096.459,131.960,-63.645,176.594,16.923,152.289
C02552=1096.453,131.711,-63.625,176.591,16.923,152.290
C02553=1096.448,131.462,-63.604,176.588,16.923,152.290
C02554=1096.442,131.213,-63.585,176.585,16.922,152.291
C02555=1096.436,130.964,-63.565,176.583,16.922,152.291
C02556=1096.430,130.715,-63.546,176.580,16.922,152.292
C02557=1096.424,130.466,-63.526,176.577,16.921,152.292
C02558=1096.419,130.216,-63.506,176.574,16.921,152.293
C02559=1096.413,129.967,-63.486,176.571,16.920,152.293
C02560=1096.408,129.718,-63.467,176.568,16.920,152.293
C02561=1096.402,129.469,-63.447,176.566,16.920,152.294
C02562=1096.396,129.219,-63.428,176.563,16.919,152.294
C02563=1096.390,128.971,-63.408,176.559,16.919,152.295
C02564=1096.385,128.721,-63.388,176.557,16.918,152.295
C02565=1096.379,128.472,-63.368,176.554,16.918,152.296
C02566=1096.372,128.197,-63.346,176.551,16.917,152.296
C02567=1096.366,127.922,-63.324,176.548,16.917,152.297
C02568=1096.360,127.646,-63.303,176.545,16.916,152.297
C02569=1096.354,127.372,-63.282,176.541,16.916,152.298
C02570=1096.348,127.123,-63.262,176.539,16.916,152.298
C02571=1096.342,126.873,-63.242,176.536,16.915,152.299
C02572=1096.336,126.624,-63.223,176.533,16.915,152.299
C02573=1096.331,126.375,-63.203,176.531,16.914,152.300
C02574=1096.325,126.125,-63.183,176.528,16.914,152.300
C02575=1096.319,125.877,-63.163,176.525,16.913,152.300
C02576=1096.314,125.628,-63.144,176.522,16.913,152.301
C02577=1096.309,125.379,-63.125,176.519,16.912,152.301
C02578=1096.303,125.130,-63.105,176.517,16.911,152.302
C02579=1096.297,124.880,-63.086,176.514,16.911,152.302
C02580=1096.291,124.631,-63.067,176.511,16.911,152.303
C02581=1096.285,124.382,-63.047,176.508,16.910,152.303
C02582=1096.280,124.133,-63.028,176.506,16.910,152.304
C02583=1096.274,123.883,-63.008,176.503,16.909,152.304
C02584=1096.270,123.634,-62.989,176.500,16.909,152.305
C02585=1096.264,123.385,-62.969,176.497,16.909,152.305
C02586=1096.258,123.136,-62.950,176.495,16.908,152.305
C02587=1096.252,122.886,-62.930,176.492,16.907,152.306
C02588=1096.247,122.637,-62.911,176.489,16.907,152.306
C02589=1096.241,122.388,-62.891,176.486,16.906,152.307
C02590=1096.235,122.139,-62.872,176.484,16.906,152.307
C02591=1096.230,121.890,-62.853,176.481,16.905,152.308
C02592=1096.224,121.641,-62.834,176.478,16.905,152.308
C02593=1096.218,121.391,-62.815,176.476,16.904,152.308
C02594=1096.212,121.142,-62.795,176.473,16.904,152.309
C02595=1096.207,120.894,-62.776,176.470,16.903,152.309
C02596=1096.202,120.644,-62.757,176.468,16.903,152.310
C02597=1096.196,120.395,-62.737,176.465,16.902,152.310
C02598=1096.190,120.145,-62.718,176.462,16.901,152.311
C02599=1096.185,119.896,-62.699,176.459,16.901,152.311
C02600=1096.179,119.647,-62.680,176.456,16.900,152.312
C02601=1096.174,119.398,-62.661,176.453,16.900,152.312
C02602=1096.168,119.149,-62.641,176.451,16.899,152.312
C02603=1096.162,118.899,-62.621,176.448,16.899,152.313
C02604=1096.157,118.651,-62.603,176.446,16.898,152.313
C02605=1096.151,118.401,-62.583,176.443,16.898,152.314
C02606=1096.146,118.152,-62.564,176.440,16.897,152.314
C02607=1096.141,117.903,-62.545,176.438,16.897,152.314
C02608=1096.135,117.654,-62.526,176.435,16.896,152.315
C02609=1096.129,117.404,-62.507,176.432,16.895,152.315
C02610=1096.123,117.155,-62.487,176.430,16.895,152.316
C02611=1096.118,116.906,-62.469,176.427,16.894,152.316
C02612=1096.113,116.657,-62.449,176.424,16.893,152.317
C02613=1096.107,116.407,-62.430,176.421,16.893,152.317
C02614=1096.101,116.159,-62.412,176.419,16.892,152.317
C02615=1096.095,115.909,-62.393,176.417,16.892,152.318
C02616=1096.090,115.660,-62.373,176.414,16.891,152.318
C02617=1096.085,115.411,-62.354,176.411,16.890,152.318
C02618=1096.079,115.162,-62.335,176.408,16.890,152.319
C02619=1096.073,114.912,-62.316,176.405,16.889,152.319
C02620=1096.068,114.664,-62.297,176.403,16.888,152.320
C02621=1096.063,114.414,-62.279,176.400,16.888,152.320
C02622=1096.057,114.164,-62.259,176.397,16.887,152.320
C02623=1096.051,113.915,-62.241,176.395,16.887,152.321
C02624=1096.046,113.666,-62.222,176.392,16.886,152.321
C02625=1096.040,113.417,-62.203,176.389,16.885,152.322
C02626=1096.034,113.167,-62.183,176.387,16.885,152.322
C02627=1096.028,112.919,-62.165,176.384,16.884,152.323
C02628=1096.023,112.670,-62.146,176.381,16.883,152.323
C02629=1096.017,112.420,-62.127,176.379,16.883,152.323
C02630=1096.011,112.145,-62.106,176.376,16.882,152.324
C02631=1096.005,111.870,-62.085,176.373,16.882,152.324
C02632=1095.999,111.595,-62.065,176.370,16.881,152.325
C02633=1095.992,111.320,-62.044,176.367,16.880,152.325
C02634=1095.987,111.070,-62.025,176.365,16.880,152.325
C02635=1095.981,110.821,-62.006,176.362,16.879,152.326
C02636=1095.976,110.572,-61.988,176.359,16.878,152.326
C02637=1095.970,110.323,-61.969,176.357,16.878,152.327
C02638=1095.964,110.073,-61.950,176.354,16.877,152.327
C02639=1095.958,109.825,-61.932,176.352,16.877,152.327
C02640=1095.953,109.575,-61.913,176.349,16.876,152.328
C02641=1095.946,109.326,-61.894,176.346,16.875,152.328
C02642=1095.941,109.077,-61.876,176.344,16.875,152.329
C02643=1095.936,108.827,-61.856,176.341,16.874,152.329
C02644=1095.930,108.578,-61.838,176.339,16.874,152.329
C02645=1095.925,108.329,-61.819,176.336,16.873,152.330
C02646=1095.919,108.079,-61.800,176.333,16.872,152.330
C02647=1095.913,107.830,-61.783,176.331,16.872,152.331
C02648=1095.908,107.581,-61.763,176.328,16.871,152.331
C02649=1095.901,107.332,-61.745,176.326,16.870,152.331
C02650=1095.896,107.083,-61.727,176.323,16.870,152.332
C02651=1095.890,106.833,-61.708,176.320,16.869,152.332
C02652=1095.885,106.584,-61.690,176.318,16.869,152.332
C02653=1095.880,106.335,-61.671,176.315,16.868,152.333
C02654=1095.873,106.086,-61.652,176.313,16.867,152.333
C02655=1095.868,105.836,-61.634,176.310,16.866,152.334
C02656=1095.862,105.587,-61.615,176.307,16.866,152.334
C02657=1095.857,105.338,-61.597,176.305,16.865,152.334
C02658=1095.851,105.089,-61.578,176.302,16.864,152.335
C02659=1095.846,104.840,-61.559,176.300,16.864,152.335
C02660=1095.839,104.590,-61.541,176.297,16.863,152.335
C02661=1095.834,104.341,-61.523,176.294,16.862,152.336
C02662=1095.828,104.092,-61.505,176.292,16.862,152.336
C02663=1095.823,103.843,-61.486,176.289,16.861,152.337
C02664=1095.817,103.593,-61.468,176.287,16.860,152.337
C02665=1095.811,103.344,-61.449,176.284,16.860,152.337
C02666=1095.807,103.094,-61.430,176.282,16.859,152.338
C02667=1095.800,102.845,-61.412,176.279,16.858,152.338
C02668=1095.795,102.596,-61.394,176.276,16.857,152.338
C02669=1095.789,102.346,-61.376,176.274,16.857,152.339
C02670=1095.784,102.097,-61.357,176.271,16.856,152.339
C02671=1095.779,101.848,-61.339,176.269,16.856,152.339
C02672=1095.772,101.599,-61.321,176.266,16.854,152.340
C02673=1095.767,101.350,-61.302,176.263,16.854,152.340
C02674=1095.761,101.101,-61.284,176.261,16.853,152.340
C02675=1095.756,100.851,-61.266,176.258,16.852,152.341
C02676=1095.750,100.602,-61.248,176.256,16.852,152.341
C02677=1095.744,100.353,-61.229,176.253,16.851,152.342
C02678=1095.739,100.103,-61.211,176.251,16.850,152.342
C02679=1095.732,99.854,-61.192,176.248,16.850,152.342
C02680=1095.727,99.605,-61.175,176.245,16.849,152.343
C02681=1095.722,99.355,-61.156,176.244,16.848,152.343
C02682=1095.716,99.107,-61.138,176.241,16.847,152.343
C02683=1095.710,98.857,-61.120,176.238,16.847,152.344
C02684=1095.705,98.607,-61.102,176.236,16.846,152.344
C02685=1095.698,98.358,-61.083,176.233,16.846,152.344
C02686=1095.693,98.109,-61.066,176.231,16.845,152.345
C02687=1095.688,97.860,-61.047,176.228,16.844,152.345
C02688=1095.682,97.610,-61.029,176.226,16.843,152.345
C02689=1095.676,97.362,-61.011,176.223,16.842,152.346
C02690=1095.670,97.112,-60.993,176.221,16.842,152.346
C02691=1095.665,96.863,-60.975,176.218,16.841,152.346
C02692=1095.659,96.614,-60.956,176.216,16.841,152.347
C02693=1095.653,96.365,-60.939,176.213,16.839,152.347
C02694=1095.647,96.089,-60.919,176.210,16.839,152.348
C02695=1095.641,95.814,-60.899,176.207,16.837,152.348
C02696=1095.634,95.539,-60.880,176.204,16.837,152.348
C02697=1095.629,95.264,-60.859,176.202,16.836,152.349
C02698=1095.623,95.014,-60.841,176.200,16.835,152.349
C02699=1095.617,94.765,-60.824,176.197,16.835,152.349
C02700=1095.611,94.516,-60.806,176.195,16.834,152.350
C02701=1095.606,94.267,-60.787,176.192,16.833,152.350
C02702=1095.601,94.018,-60.769,176.190,16.832,152.350
C02703=1095.595,93.768,-60.751,176.187,16.832,152.351
C02704=1095.589,93.519,-60.734,176.185,16.831,152.351
C02705=1095.584,93.270,-60.716,176.182,16.830,152.351
C02706=1095.578,93.020,-60.698,176.180,16.829,152.352
C02707=1095.573,92.771,-60.680,176.177,16.828,152.352
C02708=1095.567,92.521,-60.662,176.175,16.828,152.352
C02709=1095.561,92.273,-60.644,176.173,16.827,152.353
C02710=1095.555,92.024,-60.626,176.170,16.825,152.353
C02711=1095.550,91.774,-60.608,176.168,16.825,152.353
C02712=1095.544,91.525,-60.590,176.165,16.824,152.354
C02713=1095.539,91.276,-60.573,176.163,16.824,152.354
C02714=1095.533,91.026,-60.555,176.160,16.823,152.354
C02715=1095.527,90.777,-60.537,176.158,16.822,152.354
C02716=1095.522,90.528,-60.520,176.155,16.821,152.355
C02717=1095.516,90.278,-60.502,176.153,16.820,152.355
C02718=1095.510,90.029,-60.484,176.150,16.820,152.356
C02719=1095.505,89.780,-60.467,176.148,16.818,152.356
C02720=1095.498,89.530,-60.449,176.145,16.818,152.356
C02721=1095.493,89.281,-60.431,176.143,16.817,152.356
C02722=1095.487,89.032,-60.413,176.141,16.816,152.357
C02723=1095.481,88.782,-60.396,176.138,16.816,152.357
C02724=1095.476,88.533,-60.378,176.136,16.815,152.357
C02725=1095.470,88.284,-60.360,176.133,16.814,152.358
C02726=1095.464,88.035,-60.342,176.131,16.813,152.358
C02727=1095.459,87.786,-60.325,176.128,16.812,152.358
C02728=1095.453,87.536,-60.308,176.126,16.812,152.359
C02729=1095.447,87.286,-60.290,176.123,16.811,152.359
C02730=1095.442,87.037,-60.273,176.122,16.810,152.359
C02731=1095.436,86.788,-60.255,176.119,16.809,152.360
C02732=1095.430,86.538,-60.237,176.116,16.808,152.360
C02733=1095.425,86.289,-60.219,176.114,16.807,152.360
C02734=1095.419,86.040,-60.202,176.111,16.806,152.360
C02735=1095.413,85.790,-60.184,176.109,16.806,152.361
C02736=1095.408,85.541,-60.167,176.106,16.805,152.361
C02737=1095.402,85.292,-60.150,176.105,16.804,152.361
C02738=1095.397,85.043,-60.132,176.102,16.803,152.362
C02739=1095.391,84.793,-60.114,176.100,16.803,152.362
C02740=1095.385,84.544,-60.096,176.097,16.801,152.362
C02741=1095.380,84.295,-60.079,176.095,16.801,152.363
C02742=1095.374,84.045,-60.062,176.092,16.800,152.363
C02743=1095.368,83.795,-60.044,176.090,16.799,152.363
C02744=1095.363,83.546,-60.027,176.087,16.798,152.364
C02745=1095.357,83.297,-60.009,176.086,16.797,152.364
C02746=1095.352,83.048,-59.992,176.083,16.796,152.364
C02747=1095.345,82.798,-59.975,176.081,16.796,152.364
C02748=1095.340,82.549,-59.957,176.078,16.795,152.365
C02749=1095.334,82.300,-59.940,176.075,16.793,152.365
C02750=1095.329,82.051,-59.923,176.073,16.793,152.365
C02751=1095.323,81.802,-59.905,176.071,16.791,152.366
C02752=1095.317,81.552,-59.887,176.068,16.791,152.366
C02753=1095.312,81.302,-59.870,176.066,16.790,152.366
C02754=1095.306,81.053,-59.853,176.064,16.789,152.366
C02755=1095.301,80.804,-59.835,176.061,16.788,152.367
C02756=1095.296,80.554,-59.818,176.059,16.787,152.367
C02757=1095.289,80.305,-59.801,176.057,16.786,152.367
C02758=1095.283,80.030,-59.782,176.054,16.786,152.368
C02759=1095.278,79.755,-59.763,176.052,16.785,152.368
C02760=1095.271,79.480,-59.744,176.049,16.783,152.368
C02761=1095.265,79.205,-59.725,176.046,16.782,152.369
C02762=1095.260,78.956,-59.708,176.044,16.782,152.369
C02763=1095.253,78.706,-59.691,176.042,16.780,152.369
C02764=1095.247,78.457,-59.673,176.040,16.780,152.369
C02765=1095.242,78.208,-59.656,176.037,16.779,152.370
C02766=1095.237,77.958,-59.639,176.035,16.778,152.370
C02767=1095.231,77.709,-59.622,176.032,16.777,152.370
C02768=1095.225,77.460,-59.605,176.030,16.776,152.370
C02769=1095.219,77.210,-59.588,176.028,16.775,152.371
C02770=1095.213,76.961,-59.571,176.026,16.774,152.371
C02771=1095.208,76.712,-59.553,176.023,16.773,152.371
C02772=1095.202,76.462,-59.536,176.021,16.773,152.372
C02773=1095.197,76.213,-59.519,176.018,16.772,152.372
C02774=1095.191,75.964,-59.502,176.016,16.771,152.372
C02775=1095.185,75.715,-59.485,176.014,16.770,152.372
C02776=1095.180,75.465,-59.468,176.012,16.769,152.373
C02777=1095.174,75.215,-59.451,176.009,16.768,152.373
C02778=1095.168,74.966,-59.434,176.007,16.767,152.373
C02779=1095.163,74.716,-59.417,176.004,16.766,152.374
C02780=1095.157,74.468,-59.400,176.002,16.765,152.374
C02781=1095.151,74.218,-59.383,176.000,16.764,152.374
C02782=1095.146,73.969,-59.365,175.998,16.763,152.374
C02783=1095.140,73.720,-59.349,175.995,16.762,152.375
C02784=1095.134,73.470,-59.331,175.993,16.761,152.375
C02785=1095.128,73.221,-59.315,175.991,16.760,152.375
C02786=1095.123,72.971,-59.298,175.989,16.760,152.375
C02787=1095.117,72.722,-59.281,175.986,16.758,152.376
C02788=1095.111,72.473,-59.264,175.984,16.758,152.376
C02789=1095.106,72.223,-59.247,175.981,16.756,152.376
C02790=1095.100,71.974,-59.231,175.979,16.756,152.376
C02791=1095.095,71.725,-59.214,175.977,16.754,152.377
C02792=1095.089,71.475,-59.196,175.975,16.754,152.377
C02793=1095.083,71.226,-59.180,175.972,16.753,152.377
C02794=1095.078,70.976,-59.163,175.970,16.752,152.377
C02795=1095.072,70.727,-59.147,175.968,16.751,152.378
C02796=1095.066,70.478,-59.129,175.966,16.750,152.378
C02797=1095.061,70.228,-59.112,175.963,16.749,152.378
C02798=1095.055,69.979,-59.096,175.961,16.748,152.378
C02799=1095.050,69.730,-59.078,175.958,16.747,152.379
C02800=1095.043,69.480,-59.062,175.956,16.746,152.379
C02801=1095.038,69.230,-59.045,175.954,16.745,152.379
C02802=1095.032,68.981,-59.029,175.952,16.744,152.380
C02803=1095.026,68.732,-59.011,175.949,16.743,152.380
C02804=1095.021,68.483,-58.995,175.947,16.742,152.380
C02805=1095.015,68.233,-58.978,175.945,16.741,152.380
C02806=1095.009,67.984,-58.962,175.943,16.740,152.380
C02807=1095.003,67.735,-58.945,175.941,16.739,152.381
C02808=1094.998,67.485,-58.928,175.938,16.738,152.381
C02809=1094.992,67.236,-58.912,175.936,16.737,152.381
C02810=1094.987,66.986,-58.895,175.934,16.736,152.381
C02811=1094.981,66.737,-58.879,175.932,16.735,152.382
C02812=1094.976,66.487,-58.862,175.929,16.734,152.382
C02813=1094.969,66.238,-58.845,175.927,16.734,152.382
C02814=1094.963,65.989,-58.829,175.925,16.732,152.383
C02815=1094.958,65.739,-58.812,175.923,16.731,152.383
C02816=1094.952,65.490,-58.795,175.920,16.730,152.383
C02817=1094.947,65.240,-58.779,175.918,16.729,152.383
C02818=1094.941,64.991,-58.762,175.916,16.728,152.383
C02819=1094.936,64.741,-58.746,175.914,16.727,152.384
C02820=1094.930,64.493,-58.729,175.911,16.726,152.384
C02821=1094.924,64.243,-58.712,175.909,16.725,152.384
C02822=1094.918,63.968,-58.694,175.906,16.724,152.385
C02823=1094.911,63.693,-58.677,175.905,16.724,152.385
C02824=1094.904,63.418,-58.658,175.902,16.722,152.385
C02825=1094.898,63.143,-58.640,175.899,16.721,152.385
C02826=1094.892,62.893,-58.624,175.897,16.720,152.386
C02827=1094.887,62.644,-58.607,175.895,16.719,152.386
C02828=1094.881,62.394,-58.590,175.893,16.718,152.386
C02829=1094.875,62.145,-58.574,175.890,16.717,152.386
C02830=1094.869,61.896,-58.558,175.888,16.716,152.386
C02831=1094.863,61.646,-58.542,175.886,16.715,152.387
C02832=1094.857,61.397,-58.525,175.884,16.714,152.387
C02833=1094.852,61.147,-58.509,175.881,16.713,152.387
C02834=1094.846,60.898,-58.492,175.879,16.712,152.387
C02835=1094.840,60.649,-58.476,175.878,16.711,152.388
C02836=1094.834,60.399,-58.460,175.875,16.710,152.388
C02837=1094.828,60.150,-58.444,175.873,16.709,152.388
C02838=1094.823,59.900,-58.427,175.870,16.708,152.388
C02839=1094.817,59.651,-58.410,175.868,16.707,152.389
C02840=1094.812,59.402,-58.395,175.866,16.706,152.389
C02841=1094.806,59.153,-58.378,175.864,16.705,152.389
C02842=1094.800,58.904,-58.362,175.861,16.704,152.389
C02843=1094.794,58.654,-58.346,175.859,16.703,152.390
C02844=1094.789,58.405,-58.329,175.858,16.702,152.390
C02845=1094.783,58.155,-58.313,175.855,16.701,152.390
C02846=1094.777,57.905,-58.297,175.853,16.700,152.390
C02847=1094.771,57.656,-58.281,175.850,16.699,152.390
C02848=1094.765,57.407,-58.265,175.849,16.698,152.391
C02849=1094.759,57.157,-58.248,175.846,16.696,152.391
C02850=1094.753,56.908,-58.232,175.844,16.696,152.391
C02851=1094.749,56.659,-58.216,175.842,16.695,152.391
C02852=1094.743,56.409,-58.200,175.840,16.693,152.391
C02853=1094.737,56.160,-58.184,175.838,16.693,152.392
C02854=1094.731,55.910,-58.168,175.835,16.691,152.392
C02855=1094.725,55.661,-58.151,175.833,16.691,152.392
C02856=1094.719,55.412,-58.135,175.831,16.689,152.392
C02857=1094.714,55.162,-58.119,175.829,16.688,152.393
C02858=1094.708,54.913,-58.104,175.826,16.687,152.393
C02859=1094.702,54.664,-58.087,175.825,16.686,152.393
C02860=1094.697,54.414,-58.071,175.823,16.685,152.393
C02861=1094.692,54.164,-58.055,175.820,16.684,152.394
C02862=1094.686,53.915,-58.039,175.819,16.683,152.394
C02863=1094.680,53.665,-58.022,175.816,16.682,152.394
C02864=1094.674,53.417,-58.007,175.814,16.681,152.394
C02865=1094.669,53.167,-57.991,175.812,16.679,152.394
C02866=1094.663,52.917,-57.975,175.810,16.679,152.395
C02867=1094.657,52.668,-57.959,175.808,16.677,152.395
C02868=1094.651,52.418,-57.943,175.805,16.676,152.395
C02869=1094.646,52.169,-57.927,175.804,16.676,152.395
C02870=1094.640,51.920,-57.911,175.801,16.674,152.395
C02871=1094.634,51.670,-57.895,175.799,16.673,152.396
C02872=1094.628,51.421,-57.879,175.796,16.672,152.396
C02873=1094.622,51.171,-57.863,175.795,16.671,152.396
C02874=1094.618,50.922,-57.847,175.793,16.670,152.396
C02875=1094.612,50.672,-57.831,175.791,16.668,152.396
C02876=1094.606,50.423,-57.814,175.789,16.668,152.397
C02877=1094.600,50.173,-57.799,175.786,16.666,152.397
C02878=1094.595,49.924,-57.783,175.784,16.665,152.397
C02879=1094.589,49.674,-57.768,175.782,16.665,152.397
C02880=1094.584,49.425,-57.751,175.780,16.663,152.397
C02881=1094.578,49.175,-57.736,175.778,16.662,152.398
C02882=1094.573,48.927,-57.720,175.776,16.661,152.398
C02883=1094.567,48.677,-57.704,175.774,16.660,152.398
C02884=1094.561,48.427,-57.688,175.771,16.658,152.398
C02885=1094.556,48.179,-57.672,175.770,16.658,152.398
C02886=1094.548,47.902,-57.655,175.767,16.656,152.398
C02887=1094.542,47.627,-57.637,175.765,16.655,152.399
C02888=1094.536,47.352,-57.620,175.763,16.653,152.399
C02889=1094.531,47.076,-57.602,175.760,16.652,152.399
C02890=1094.525,46.828,-57.587,175.758,16.652,152.399
C02891=1094.520,46.578,-57.571,175.757,16.650,152.399
C02892=1094.514,46.328,-57.555,175.754,16.649,152.400
C02893=1094.509,46.079,-57.540,175.752,16.648,152.400
C02894=1094.502,45.830,-57.524,175.750,16.646,152.400
C02895=1094.496,45.580,-57.508,175.748,16.646,152.400
C02896=1094.491,45.331,-57.493,175.746,16.644,152.400
C02897=1094.485,45.082,-57.477,175.744,16.643,152.401
C02898=1094.480,44.832,-57.461,175.742,16.642,152.401
C02899=1094.474,44.583,-57.445,175.739,16.641,152.401
C02900=1094.469,44.333,-57.430,175.738,16.640,152.401
C02901=1094.463,44.083,-57.414,175.735,16.638,152.401
C02902=1094.458,43.834,-57.399,175.733,16.637,152.401
C02903=1094.452,43.584,-57.383,175.732,16.636,152.402
C02904=1094.446,43.335,-57.367,175.729,16.635,152.402
C02905=1094.440,43.086,-57.352,175.727,16.634,152.402
C02906=1094.435,42.836,-57.337,175.725,16.633,152.402
C02907=1094.429,42.587,-57.320,175.723,16.631,152.402
C02908=1094.424,42.338,-57.305,175.721,16.631,152.403
C02909=1094.418,42.088,-57.290,175.719,16.629,152.403
C02910=1094.411,41.839,-57.274,175.717,16.628,152.403
C02911=1094.406,41.589,-57.259,175.715,16.627,152.403
C02912=1094.401,41.339,-57.243,175.713,16.626,152.403
C02913=1094.395,41.090,-57.227,175.711,16.625,152.403
C02914=1094.389,40.841,-57.212,175.708,16.624,152.404
C02915=1094.383,40.591,-57.197,175.707,16.622,152.404
C02916=1094.377,40.342,-57.181,175.705,16.622,152.404
C02917=1094.372,40.092,-57.165,175.702,16.620,152.404
C02918=1094.366,39.843,-57.150,175.701,16.619,152.404
C02919=1094.361,39.593,-57.135,175.698,16.618,152.405
C02920=1094.355,39.344,-57.119,175.696,16.617,152.405
C02921=1094.349,39.094,-57.104,175.695,16.616,152.405
C02922=1094.343,38.845,-57.089,175.692,16.614,152.405
C02923=1094.338,38.595,-57.073,175.691,16.613,152.405
C02924=1094.332,38.347,-57.057,175.689,16.612,152.405
C02925=1094.327,38.097,-57.042,175.686,16.611,152.405
C02926=1094.320,37.847,-57.027,175.684,16.610,152.406
C02927=1094.315,37.598,-57.012,175.682,16.608,152.406
C02928=1094.309,37.348,-56.997,175.680,16.607,152.406
C02929=1094.304,37.099,-56.981,175.678,16.606,152.406
C02930=1094.298,36.849,-56.965,175.676,16.605,152.406
C02931=1094.292,36.600,-56.951,175.674,16.604,152.407
C02932=1094.287,36.350,-56.935,175.673,16.603,152.407
C02933=1094.280,36.101,-56.920,175.670,16.602,152.407
C02934=1094.275,35.852,-56.905,175.668,16.600,152.407
C02935=1094.269,35.602,-56.890,175.666,16.599,152.407
C02936=1094.263,35.353,-56.874,175.664,16.598,152.407
C02937=1094.258,35.103,-56.859,175.662,16.597,152.408
C02938=1094.251,34.854,-56.844,175.660,16.596,152.408
C02939=1094.246,34.604,-56.829,175.658,16.595,152.408
C02940=1094.240,34.355,-56.814,175.656,16.593,152.408
C02941=1094.234,34.105,-56.798,175.654,16.592,152.408
C02942=1094.229,33.856,-56.784,175.652,16.591,152.408
C02943=1094.223,33.606,-56.768,175.650,16.590,152.408
C02944=1094.218,33.357,-56.753,175.648,16.589,152.409
C02945=1094.211,33.107,-56.738,175.646,16.588,152.409
C02946=1094.206,32.858,-56.723,175.644,16.586,152.409
C02947=1094.200,32.608,-56.708,175.642,16.585,152.409
C02948=1094.195,32.359,-56.693,175.640,16.584,152.409
C02949=1094.189,32.109,-56.678,175.638,16.582,152.409
C02950=1094.182,31.834,-56.660,175.636,16.582,152.410
C02951=1094.175,31.559,-56.644,175.633,16.580,152.410
C02952=1094.170,31.284,-56.627,175.632,16.579,152.410
C02953=1094.164,31.008,-56.611,175.629,16.578,152.410
C02954=1094.157,30.759,-56.596,175.628,16.576,152.410
C02955=1094.152,30.509,-56.581,175.625,16.575,152.410
C02956=1094.146,30.260,-56.566,175.623,16.574,152.411
C02957=1094.141,30.010,-56.550,175.622,16.573,152.411
C02958=1094.134,29.761,-56.535,175.619,16.571,152.411
C02959=1094.129,29.512,-56.520,175.617,16.570,152.411
C02960=1094.123,29.261,-56.506,175.616,16.569,152.411
C02961=1094.118,29.012,-56.491,175.613,16.568,152.411
C02962=1094.112,28.762,-56.476,175.612,16.566,152.412
C02963=1094.107,28.513,-56.461,175.610,16.566,152.412
C02964=1094.100,28.263,-56.446,175.607,16.564,152.412
C02965=1094.095,28.014,-56.431,175.606,16.563,152.412
C02966=1094.089,27.764,-56.416,175.604,16.562,152.412
C02967=1094.083,27.516,-56.401,175.601,16.561,152.412
C02968=1094.077,27.267,-56.387,175.600,16.559,152.412
C02969=1094.072,27.016,-56.372,175.598,16.559,152.413
C02970=1094.066,26.767,-56.357,175.596,16.557,152.413
C02971=1094.060,26.517,-56.342,175.594,16.556,152.413
C02972=1094.055,26.268,-56.327,175.592,16.555,152.413
C02973=1094.048,26.018,-56.312,175.590,16.553,152.413
C02974=1094.043,25.770,-56.297,175.588,16.552,152.413
C02975=1094.037,25.519,-56.283,175.586,16.551,152.414
C02976=1094.032,25.270,-56.268,175.584,16.550,152.414
C02977=1094.025,25.020,-56.253,175.582,16.549,152.414
C02978=1094.020,24.771,-56.238,175.580,16.548,152.414
C02979=1094.014,24.521,-56.223,175.578,16.546,152.414
C02980=1094.008,24.272,-56.209,175.576,16.545,152.414
C02981=1094.003,24.023,-56.194,175.575,16.544,152.414
C02982=1093.997,23.773,-56.179,175.572,16.542,152.415
C02983=1093.991,23.524,-56.164,175.570,16.541,152.415
C02984=1093.985,23.274,-56.150,175.569,16.541,152.415
C02985=1093.980,23.024,-56.135,175.566,16.539,152.415
C02986=1093.974,22.775,-56.120,175.565,16.538,152.415
C02987=1093.968,22.525,-56.106,175.563,16.537,152.415
C02988=1093.962,22.276,-56.092,175.560,16.535,152.416
C02989=1093.957,22.026,-56.076,175.559,16.534,152.416
C02990=1093.951,21.777,-56.062,175.557,16.533,152.416
C02991=1093.945,21.527,-56.047,175.555,16.531,152.416
C02992=1093.939,21.278,-56.033,175.553,16.530,152.416
C02993=1093.934,21.029,-56.018,175.551,16.530,152.416
C02994=1093.928,20.779,-56.003,175.549,16.528,152.416
C02995=1093.922,20.530,-55.989,175.547,16.527,152.417
C02996=1093.917,20.280,-55.975,175.545,16.526,152.417
C02997=1093.911,20.030,-55.959,175.543,16.524,152.417
C02998=1093.905,19.781,-55.945,175.541,16.523,152.417
C02999=1093.899,19.531,-55.931,175.540,16.522,152.417
C03000=1093.893,19.282,-55.916,175.538,16.521,152.417
C03001=1093.888,19.033,-55.901,175.536,16.519,152.417
C03002=1093.882,18.783,-55.887,175.534,16.518,152.417
C03003=1093.876,18.533,-55.872,175.532,16.517,152.418
C03004=1093.871,18.284,-55.858,175.530,16.516,152.418
C03005=1093.865,18.034,-55.843,175.528,16.514,152.418
C03006=1093.859,17.785,-55.829,175.526,16.513,152.418
C03007=1093.853,17.535,-55.814,175.524,16.512,152.418
C03008=1093.847,17.286,-55.800,175.522,16.511,152.418
C03009=1093.842,17.036,-55.786,175.520,16.510,152.418
C03010=1093.835,16.787,-55.771,175.519,16.509,152.419
C03011=1093.830,16.537,-55.756,175.516,16.507,152.419
C03012=1093.825,16.288,-55.742,175.515,16.506,152.419
C03013=1093.819,16.038,-55.728,175.513,16.505,152.419
C03014=1093.812,15.764,-55.712,175.511,16.503,152.419
C03015=1093.806,15.490,-55.696,175.509,16.502,152.419
C03016=1093.800,15.216,-55.681,175.507,16.501,152.419
C03017=1093.794,14.943,-55.664,175.505,16.499,152.420
C03018=1093.788,14.693,-55.650,175.502,16.498,152.420
C03019=1093.782,14.444,-55.636,175.501,16.497,152.420
C03020=1093.777,14.194,-55.622,175.499,16.495,152.420
C03021=1093.770,13.945,-55.607,175.497,16.494,152.420
C03022=1093.765,13.695,-55.593,175.495,16.493,152.420
C03023=1093.759,13.445,-55.579,175.493,16.492,152.420
C03024=1093.753,13.196,-55.564,175.492,16.491,152.420
C03025=1093.747,12.946,-55.551,175.489,16.489,152.421
C03026=1093.741,12.697,-55.536,175.487,16.488,152.421
C03027=1093.735,12.447,-55.522,175.486,16.487,152.421
C03028=1093.729,12.198,-55.508,175.483,16.485,152.421
C03029=1093.724,11.949,-55.494,175.482,16.484,152.421
C03030=1093.717,11.698,-55.479,175.480,16.483,152.421
C03031=1093.712,11.449,-55.465,175.478,16.483,152.422
C03032=1093.706,11.200,-55.451,175.476,16.481,152.422
C03033=1093.700,10.950,-55.437,175.474,16.480,152.422
C03034=1093.694,10.701,-55.422,175.473,16.478,152.422
C03035=1093.689,10.451,-55.408,175.471,16.477,152.422
C03036=1093.683,10.202,-55.395,175.469,16.476,152.422
C03037=1093.676,9.952,-55.380,175.467,16.475,152.422
C03038=1093.671,9.703,-55.366,175.465,16.474,152.422
C03039=1093.665,9.453,-55.352,175.463,16.472,152.423
C03040=1093.659,9.203,-55.337,175.461,16.471,152.423
C03041=1093.653,8.954,-55.324,175.459,16.470,152.423
C03042=1093.648,8.704,-55.310,175.458,16.469,152.423
C03043=1093.642,8.455,-55.296,175.455,16.467,152.423
C03044=1093.635,8.205,-55.281,175.454,16.466,152.423
C03045=1093.630,7.956,-55.268,175.452,16.465,152.423
C03046=1093.624,7.706,-55.254,175.450,16.464,152.423
C03047=1093.619,7.457,-55.240,175.448,16.462,152.424
C03048=1093.613,7.207,-55.225,175.446,16.461,152.424
C03049=1093.607,6.957,-55.211,175.445,16.460,152.424
C03050=1093.602,6.708,-55.197,175.443,16.459,152.424
C03051=1093.595,6.458,-55.184,175.441,16.457,152.424
C03052=1093.590,6.210,-55.169,175.439,16.456,152.424
C03053=1093.584,5.959,-55.155,175.437,16.455,152.424
C03054=1093.578,5.710,-55.141,175.436,16.454,152.424
C03055=1093.573,5.460,-55.127,175.433,16.452,152.425
C03056=1093.567,5.211,-55.114,175.432,16.451,152.425
C03057=1093.561,4.962,-55.100,175.430,16.450,152.425
C03058=1093.554,4.712,-55.085,175.428,16.449,152.425
C03059=1093.549,4.462,-55.071,175.426,16.447,152.425
C03060=1093.544,4.212,-55.058,175.424,16.446,152.425
C03061=1093.538,3.963,-55.044,175.423,16.445,152.425
C03062=1093.532,3.714,-55.030,175.421,16.444,152.425
C03063=1093.526,3.464,-55.017,175.419,16.442,152.425
C03064=1093.520,3.214,-55.002,175.417,16.441,152.426
C03065=1093.515,2.965,-54.988,175.415,16.440,152.426
C03066=1093.509,2.715,-54.974,175.414,16.439,152.426
C03067=1093.503,2.466,-54.961,175.411,16.437,152.426
C03068=1093.497,2.216,-54.947,175.410,16.436,152.426
C03069=1093.492,1.967,-54.933,175.408,16.435,152.426
C03070=1093.486,1.717,-54.919,175.406,16.434,152.426
C03071=1093.480,1.467,-54.905,175.404,16.432,152.426
C03072=1093.474,1.218,-54.892,175.402,16.431,152.427
C03073=1093.469,0.968,-54.878,175.401,16.430,152.427
C03074=1093.463,0.719,-54.864,175.399,16.429,152.427
C03075=1093.458,0.469,-54.850,175.397,16.427,152.427
C03076=1093.451,0.220,-54.837,175.395,16.426,152.427
C03077=1093.446,-0.030,-54.823,175.393,16.425,152.427
C03078=1093.440,-0.302,-54.808,175.391,16.423,152.427
C03079=1093.433,-0.574,-54.793,175.389,16.422,152.427
C03080=1093.427,-0.845,-54.778,175.388,16.421,152.427
C03081=1093.421,-1.118,-54.763,175.385,16.419,152.428
C03082=1093.415,-1.367,-54.749,175.384,16.418,152.428
C03083=1093.410,-1.616,-54.736,175.382,16.417,152.428
C03084=1093.404,-1.866,-54.722,175.380,16.415,152.428
C03085=1093.398,-2.115,-54.708,175.378,16.414,152.428
C03086=1093.393,-2.365,-54.695,175.377,16.413,152.428
C03087=1093.387,-2.614,-54.681,175.375,16.412,152.428
C03088=1093.381,-2.865,-54.666,175.373,16.410,152.428
C03089=1093.375,-3.114,-54.653,175.371,16.409,152.428
C03090=1093.369,-3.364,-54.639,175.369,16.408,152.429
C03091=1093.364,-3.613,-54.625,175.368,16.406,152.429
C03092=1093.358,-3.863,-54.613,175.366,16.405,152.429
C03093=1093.352,-4.113,-54.599,175.364,16.404,152.429
C03094=1093.346,-4.362,-54.586,175.362,16.402,152.429
C03095=1093.341,-4.611,-54.572,175.360,16.401,152.429
C03096=1093.335,-4.861,-54.559,175.359,16.400,152.429
C03097=1093.329,-5.110,-54.545,175.357,16.399,152.429
C03098=1093.323,-5.360,-54.532,175.355,16.397,152.429
C03099=1093.317,-5.610,-54.517,175.353,16.396,152.430
C03100=1093.311,-5.860,-54.505,175.351,16.395,152.430
C03101=1093.305,-6.109,-54.491,175.350,16.394,152.430
C03102=1093.299,-6.359,-54.478,175.347,16.393,152.430
C03103=1093.294,-6.608,-54.464,175.346,16.391,152.430
C03104=1093.287,-6.857,-54.450,175.344,16.390,152.430
C03105=1093.282,-7.107,-54.437,175.342,16.389,152.430
C03106=1093.276,-7.357,-54.424,175.341,16.388,152.430
C03107=1093.270,-7.606,-54.411,175.338,16.386,152.431
C03108=1093.264,-7.856,-54.397,175.337,16.385,152.431
C03109=1093.258,-8.105,-54.384,175.335,16.384,152.431
C03110=1093.253,-8.355,-54.370,175.334,16.383,152.431
C03111=1093.247,-8.604,-54.357,175.332,16.382,152.431
C03112=1093.241,-8.854,-54.343,175.330,16.380,152.431
C03113=1093.235,-9.103,-54.330,175.328,16.379,152.431
C03114=1093.230,-9.353,-54.316,175.326,16.378,152.431
C03115=1093.224,-9.603,-54.304,175.325,16.377,152.431
C03116=1093.218,-9.852,-54.290,175.323,16.375,152.431
C03117=1093.212,-10.102,-54.277,175.321,16.374,152.432
C03118=1093.206,-10.351,-54.264,175.319,16.373,152.432
C03119=1093.201,-10.601,-54.250,175.318,16.371,152.432
C03120=1093.194,-10.850,-54.237,175.316,16.370,152.432
C03121=1093.189,-11.100,-54.224,175.314,16.369,152.432
C03122=1093.183,-11.350,-54.210,175.312,16.367,152.432
C03123=1093.178,-11.599,-54.197,175.310,16.366,152.432
C03124=1093.172,-11.849,-54.184,175.309,16.365,152.432
C03125=1093.165,-12.098,-54.171,175.307,16.364,152.432
C03126=1093.160,-12.348,-54.157,175.305,16.363,152.433
C03127=1093.154,-12.598,-54.144,175.303,16.361,152.433
C03128=1093.149,-12.847,-54.130,175.301,16.360,152.433
C03129=1093.142,-13.097,-54.117,175.300,16.359,152.433
C03130=1093.136,-13.347,-54.105,175.298,16.358,152.433
C03131=1093.131,-13.596,-54.091,175.297,16.357,152.433
C03132=1093.125,-13.845,-54.078,175.295,16.355,152.433
C03133=1093.120,-14.096,-54.064,175.293,16.354,152.433
C03134=1093.113,-14.345,-54.051,175.291,16.352,152.433
C03135=1093.107,-14.595,-54.039,175.289,16.351,152.434
C03136=1093.102,-14.844,-54.025,175.288,16.350,152.434
C03137=1093.096,-15.094,-54.012,175.286,16.349,152.434
C03138=1093.090,-15.344,-53.999,175.284,16.347,152.434
C03139=1093.084,-15.593,-53.985,175.282,16.346,152.434
C03140=1093.079,-15.842,-53.973,175.281,16.345,152.434
C03141=1093.073,-16.092,-53.960,175.279,16.344,152.434
C03142=1093.066,-16.363,-53.946,175.277,16.343,152.434
C03143=1093.060,-16.632,-53.931,175.275,16.341,152.434
C03144=1093.054,-16.903,-53.918,175.273,16.340,152.435
C03145=1093.047,-17.173,-53.903,175.272,16.339,152.435
C03146=1093.041,-17.423,-53.890,175.269,16.337,152.435
C03147=1093.035,-17.672,-53.877,175.267,16.336,152.435
C03148=1093.030,-17.922,-53.864,175.266,16.335,152.435
C03149=1093.023,-18.172,-53.851,175.264,16.334,152.435
C03150=1093.018,-18.421,-53.838,175.263,16.333,152.435
C03151=1093.012,-18.670,-53.825,175.261,16.332,152.435
C03152=1093.006,-18.920,-53.813,175.259,16.330,152.436
C03153=1093.001,-19.170,-53.799,175.257,16.329,152.436
C03154=1092.995,-19.419,-53.786,175.255,16.328,152.436
C03155=1092.989,-19.669,-53.774,175.254,16.327,152.436
C03156=1092.983,-19.918,-53.760,175.252,16.325,152.436
C03157=1092.977,-20.168,-53.748,175.251,16.324,152.436
C03158=1092.971,-20.418,-53.734,175.248,16.323,152.436
C03159=1092.965,-20.668,-53.721,175.247,16.321,152.436
C03160=1092.960,-20.917,-53.709,175.245,16.320,152.436
C03161=1092.954,-21.166,-53.696,175.243,16.319,152.437
C03162=1092.948,-21.416,-53.683,175.242,16.318,152.437
C03163=1092.942,-21.665,-53.670,175.240,16.317,152.437
C03164=1092.936,-21.915,-53.658,175.238,16.316,152.437
C03165=1092.930,-22.165,-53.644,175.236,16.314,152.437
C03166=1092.924,-22.415,-53.631,175.234,16.313,152.437
C03167=1092.918,-22.665,-53.619,175.233,16.312,152.437
C03168=1092.913,-22.914,-53.606,175.231,16.311,152.437
C03169=1092.907,-23.163,-53.593,175.230,16.309,152.437
C03170=1092.901,-23.413,-53.581,175.228,16.308,152.437
C03171=1092.895,-23.663,-53.568,175.226,16.307,152.438
C03172=1092.890,-23.912,-53.554,175.224,16.305,152.438
C03173=1092.884,-24.162,-53.542,175.222,16.304,152.438
C03174=1092.878,-24.411,-53.529,175.221,16.303,152.438
C03175=1092.872,-24.661,-53.516,175.219,16.302,152.438
C03176=1092.866,-24.911,-53.504,175.218,16.301,152.438
C03177=1092.860,-25.161,-53.491,175.216,16.300,152.438
C03178=1092.854,-25.410,-53.478,175.214,16.299,152.438
C03179=1092.849,-25.659,-53.466,175.212,16.297,152.438
C03180=1092.843,-25.909,-53.453,175.210,16.296,152.439
C03181=1092.837,-26.159,-53.440,175.209,16.295,152.439
C03182=1092.832,-26.409,-53.427,175.207,16.293,152.439
C03183=1092.826,-26.658,-53.414,175.206,16.292,152.439
C03184=1092.820,-26.907,-53.402,175.204,16.291,152.439
C03185=1092.814,-27.157,-53.389,175.202,16.290,152.439
C03186=1092.808,-27.407,-53.377,175.201,16.289,152.439
C03187=1092.802,-27.656,-53.363,175.198,16.287,152.439
C03188=1092.796,-27.906,-53.351,175.197,16.286,152.439
C03189=1092.790,-28.155,-53.339,175.195,16.285,152.440
C03190=1092.784,-28.405,-53.327,175.193,16.284,152.440
C03191=1092.778,-28.655,-53.314,175.192,16.282,152.440
C03192=1092.772,-28.904,-53.301,175.190,16.281,152.440
C03193=1092.766,-29.154,-53.288,175.189,16.280,152.440
C03194=1092.760,-29.404,-53.276,175.187,16.279,152.440
C03195=1092.755,-29.653,-53.264,175.185,16.278,152.440
C03196=1092.749,-29.903,-53.251,175.183,16.276,152.440
C03197=1092.743,-30.153,-53.239,175.181,16.275,152.440
C03198=1092.737,-30.403,-53.226,175.180,16.274,152.440
C03199=1092.731,-30.652,-53.213,175.178,16.273,152.441
C03200=1092.725,-30.901,-53.201,175.177,16.272,152.441
C03201=1092.719,-31.151,-53.189,175.175,16.270,152.441
C03202=1092.713,-31.401,-53.176,175.173,16.269,152.441
C03203=1092.707,-31.651,-53.163,175.172,16.268,152.441
C03204=1092.702,-31.900,-53.151,175.170,16.267,152.441
C03205=1092.696,-32.150,-53.139,175.168,16.265,152.441
C03206=1092.689,-32.419,-53.125,175.166,16.264,152.441
C03207=1092.684,-32.689,-53.112,175.165,16.263,152.441
C03208=1092.677,-32.958,-53.098,175.163,16.262,152.442
C03209=1092.670,-33.227,-53.085,175.160,16.260,152.442
C03210=1092.665,-33.477,-53.073,175.159,16.259,152.442
C03211=1092.659,-33.726,-53.061,175.157,16.258,152.442
C03212=1092.653,-33.976,-53.048,175.155,16.257,152.442
C03213=1092.647,-34.226,-53.035,175.154,16.256,152.442
C03214=1092.642,-34.476,-53.023,175.152,16.255,152.442
C03215=1092.635,-34.725,-53.011,175.151,16.254,152.442
C03216=1092.630,-34.975,-52.999,175.149,16.253,152.443
C03217=1092.624,-35.225,-52.986,175.147,16.251,152.443
C03218=1092.618,-35.474,-52.974,175.146,16.250,152.443
C03219=1092.612,-35.724,-52.961,175.143,16.249,152.443
C03220=1092.607,-35.974,-52.949,175.142,16.247,152.443
C03221=1092.600,-36.223,-52.937,175.140,16.246,152.443
C03222=1092.595,-36.472,-52.925,175.138,16.245,152.443
C03223=1092.589,-36.722,-52.912,175.137,16.244,152.443
C03224=1092.583,-36.972,-52.900,175.135,16.243,152.443
C03225=1092.577,-37.221,-52.887,175.134,16.242,152.444
C03226=1092.572,-37.471,-52.875,175.132,16.241,152.444
C03227=1092.565,-37.721,-52.863,175.130,16.239,152.444
C03228=1092.560,-37.970,-52.851,175.129,16.238,152.444
C03229=1092.554,-38.220,-52.838,175.127,16.237,152.444
C03230=1092.548,-38.470,-52.826,175.126,16.236,152.444
C03231=1092.542,-38.719,-52.813,175.123,16.234,152.444
C03232=1092.536,-38.969,-52.802,175.122,16.233,152.444
C03233=1092.530,-39.219,-52.790,175.120,16.232,152.444
C03234=1092.525,-39.468,-52.777,175.118,16.231,152.444
C03235=1092.518,-39.718,-52.765,175.117,16.230,152.445
C03236=1092.512,-39.968,-52.753,175.115,16.229,152.445
C03237=1092.506,-40.216,-52.741,175.114,16.227,152.445
C03238=1092.500,-40.466,-52.729,175.112,16.226,152.445
C03239=1092.495,-40.716,-52.716,175.110,16.225,152.445
C03240=1092.489,-40.966,-52.705,175.108,16.224,152.445
C03241=1092.483,-41.216,-52.693,175.107,16.223,152.445
C03242=1092.477,-41.465,-52.680,175.105,16.222,152.445
C03243=1092.471,-41.714,-52.669,175.104,16.221,152.446
C03244=1092.465,-41.964,-52.656,175.102,16.220,152.446
C03245=1092.459,-42.214,-52.644,175.100,16.219,152.446
C03246=1092.453,-42.464,-52.633,175.099,16.218,152.446
C03247=1092.447,-42.713,-52.620,175.096,16.216,152.446
C03248=1092.441,-42.963,-52.608,175.095,16.215,152.446
C03249=1092.435,-43.212,-52.596,175.093,16.214,152.446
C03250=1092.430,-43.463,-52.584,175.092,16.212,152.446
C03251=1092.424,-43.712,-52.573,175.090,16.211,152.446
C03252=1092.418,-43.961,-52.560,175.088,16.210,152.447
C03253=1092.411,-44.211,-52.548,175.087,16.209,152.447
C03254=1092.406,-44.461,-52.537,175.085,16.208,152.447
C03255=1092.400,-44.711,-52.524,175.083,16.207,152.447
C03256=1092.394,-44.960,-52.512,175.082,16.206,152.447
C03257=1092.388,-45.209,-52.500,175.080,16.205,152.447
C03258=1092.382,-45.460,-52.489,175.078,16.204,152.447
C03259=1092.377,-45.709,-52.476,175.077,16.203,152.447
C03260=1092.370,-45.958,-52.464,175.075,16.201,152.448
C03261=1092.364,-46.208,-52.452,175.074,16.200,152.448
C03262=1092.359,-46.458,-52.440,175.072,16.199,152.448
C03263=1092.353,-46.708,-52.428,175.070,16.198,152.448
C03264=1092.347,-46.957,-52.416,175.069,16.197,152.448
C03265=1092.341,-47.207,-52.405,175.067,16.196,152.448
C03266=1092.336,-47.456,-52.393,175.066,16.195,152.448
C03267=1092.329,-47.706,-52.381,175.064,16.193,152.448
C03268=1092.323,-47.956,-52.369,175.062,16.193,152.448
C03269=1092.317,-48.205,-52.357,175.060,16.192,152.449
C03270=1092.311,-48.475,-52.344,175.058,16.190,152.449
C03271=1092.305,-48.745,-52.332,175.056,16.189,152.449
C03272=1092.299,-49.015,-52.319,175.055,16.188,152.449
C03273=1092.292,-49.285,-52.306,175.053,16.186,152.449
C03274=1092.286,-49.534,-52.294,175.052,16.185,152.449
C03275=1092.281,-49.784,-52.283,175.050,16.184,152.449
C03276=1092.274,-50.034,-52.271,175.048,16.183,152.449
C03277=1092.269,-50.283,-52.259,175.047,16.182,152.449
C03278=1092.263,-50.533,-52.247,175.045,16.181,152.450
C03279=1092.257,-50.782,-52.235,175.044,16.180,152.450
C03280=1092.251,-51.032,-52.224,175.042,16.179,152.450
C03281=1092.245,-51.281,-52.212,175.040,16.178,152.450
C03282=1092.239,-51.532,-52.200,175.038,16.177,152.450
C03283=1092.233,-51.781,-52.189,175.037,16.175,152.450
C03284=1092.227,-52.031,-52.178,175.035,16.174,152.450
C03285=1092.220,-52.280,-52.166,175.033,16.174,152.451
C03286=1092.215,-52.529,-52.153,175.032,16.173,152.451
C03287=1092.209,-52.780,-52.142,175.030,16.171,152.451
C03288=1092.202,-53.029,-52.130,175.029,16.170,152.451
C03289=1092.197,-53.279,-52.119,175.027,16.169,152.451
C03290=1092.190,-53.529,-52.107,175.025,16.168,152.451
C03291=1092.185,-53.778,-52.096,175.023,16.167,152.451
C03292=1092.178,-54.028,-52.084,175.022,16.166,152.452
C03293=1092.173,-54.277,-52.073,175.020,16.165,152.452
C03294=1092.166,-54.527,-52.061,175.019,16.164,152.452
C03295=1092.161,-54.777,-52.050,175.017,16.163,152.452
C03296=1092.154,-55.026,-52.038,175.015,16.162,152.452
C03297=1092.148,-55.277,-52.026,175.013,16.161,152.452
C03298=1092.142,-55.525,-52.014,175.012,16.160,152.452
C03299=1092.136,-55.776,-52.003,175.010,16.159,152.452
C03300=1092.130,-56.025,-51.992,175.009,16.158,152.452
C03301=1092.124,-56.275,-51.980,175.007,16.156,152.453
C03302=1092.118,-56.525,-51.969,175.005,16.156,152.453
C03303=1092.112,-56.774,-51.957,175.004,16.155,152.453
C03304=1092.106,-57.024,-51.946,175.002,16.153,152.453
C03305=1092.100,-57.273,-51.933,175.000,16.152,152.453
C03306=1092.094,-57.523,-51.922,174.999,16.151,152.453
C03307=1092.088,-57.773,-51.911,174.997,16.150,152.454
C03308=1092.082,-58.022,-51.900,174.995,16.149,152.454
C03309=1092.076,-58.273,-51.888,174.994,16.148,152.454
C03310=1092.071,-58.522,-51.877,174.992,16.147,152.454
C03311=1092.064,-58.772,-51.865,174.990,16.146,152.454
C03312=1092.058,-59.021,-51.854,174.988,16.145,152.454
C03313=1092.052,-59.271,-51.842,174.987,16.144,152.454
C03314=1092.047,-59.520,-51.831,174.985,16.143,152.454
C03315=1092.040,-59.771,-51.819,174.984,16.142,152.455
C03316=1092.034,-60.020,-51.808,174.982,16.141,152.455
C03317=1092.029,-60.269,-51.797,174.980,16.140,152.455
C03318=1092.022,-60.519,-51.786,174.979,16.139,152.455
C03319=1092.017,-60.768,-51.774,174.977,16.138,152.455
C03320=1092.011,-61.019,-51.762,174.975,16.137,152.455
C03321=1092.005,-61.268,-51.751,174.974,16.135,152.455
C03322=1091.999,-61.518,-51.740,174.972,16.134,152.455
C03323=1091.992,-61.767,-51.729,174.971,16.134,152.456
C03324=1091.986,-62.017,-51.717,174.969,16.133,152.456
C03325=1091.981,-62.267,-51.706,174.968,16.132,152.456
C03326=1091.975,-62.516,-51.694,174.966,16.131,152.456
C03327=1091.969,-62.766,-51.683,174.965,16.130,152.456
C03328=1091.963,-63.016,-51.672,174.963,16.129,152.456
C03329=1091.957,-63.266,-51.661,174.961,16.128,152.456
C03330=1091.951,-63.515,-51.649,174.959,16.127,152.457
C03331=1091.946,-63.765,-51.638,174.958,16.126,152.457
C03332=1091.939,-64.015,-51.627,174.956,16.124,152.457
C03333=1091.934,-64.264,-51.616,174.954,16.124,152.457
C03334=1091.927,-64.535,-51.603,174.953,16.123,152.457
C03335=1091.920,-64.807,-51.591,174.951,16.121,152.457
C03336=1091.914,-65.077,-51.579,174.950,16.120,152.457
C03337=1091.907,-65.348,-51.567,174.948,16.120,152.458
C03338=1091.901,-65.598,-51.556,174.946,16.119,152.458
C03339=1091.895,-65.848,-51.545,174.944,16.117,152.458
C03340=1091.890,-66.098,-51.533,174.943,16.116,152.458
C03341=1091.884,-66.348,-51.522,174.941,16.115,152.458
C03342=1091.878,-66.597,-51.511,174.939,16.114,152.458
C03343=1091.872,-66.846,-51.499,174.938,16.113,152.458
C03344=1091.866,-67.096,-51.488,174.936,16.112,152.458
C03345=1091.860,-67.346,-51.477,174.934,16.111,152.459
C03346=1091.854,-67.595,-51.466,174.933,16.110,152.459
C03347=1091.848,-67.845,-51.455,174.931,16.109,152.459
C03348=1091.842,-68.095,-51.444,174.929,16.108,152.459
C03349=1091.837,-68.344,-51.433,174.928,16.107,152.459
C03350=1091.831,-68.595,-51.422,174.927,16.106,152.459
C03351=1091.825,-68.844,-51.410,174.925,16.106,152.459
C03352=1091.819,-69.093,-51.399,174.923,16.105,152.460
C03353=1091.813,-69.343,-51.388,174.922,16.103,152.460
C03354=1091.807,-69.593,-51.377,174.920,16.102,152.460
C03355=1091.801,-69.842,-51.366,174.919,16.101,152.460
C03356=1091.795,-70.093,-51.355,174.917,16.101,152.460
C03357=1091.789,-70.342,-51.344,174.915,16.099,152.460
C03358=1091.784,-70.592,-51.333,174.913,16.098,152.460
C03359=1091.778,-70.841,-51.322,174.912,16.097,152.461
C03360=1091.771,-71.091,-51.311,174.910,16.096,152.461
C03361=1091.766,-71.341,-51.300,174.908,16.095,152.461
C03362=1091.760,-71.590,-51.289,174.908,16.095,152.461
C03363=1091.754,-71.840,-51.278,174.906,16.094,152.461
C03364=1091.749,-72.090,-51.267,174.904,16.092,152.461
C03365=1091.743,-72.340,-51.256,174.902,16.092,152.461
C03366=1091.737,-72.589,-51.245,174.901,16.091,152.462
C03367=1091.731,-72.839,-51.234,174.899,16.089,152.462
C03368=1091.725,-73.089,-51.223,174.898,16.088,152.462
C03369=1091.719,-73.338,-51.212,174.896,16.088,152.462
C03370=1091.714,-73.588,-51.201,174.894,16.087,152.462
C03371=1091.707,-73.838,-51.190,174.892,16.085,152.462
C03372=1091.702,-74.088,-51.179,174.892,16.085,152.462
C03373=1091.696,-74.337,-51.168,174.890,16.084,152.463
C03374=1091.690,-74.587,-51.157,174.888,16.083,152.463
C03375=1091.683,-74.836,-51.146,174.887,16.082,152.463
C03376=1091.677,-75.086,-51.136,174.885,16.081,152.463
C03377=1091.671,-75.335,-51.125,174.883,16.080,152.463
C03378=1091.665,-75.586,-51.113,174.881,16.079,152.463
C03379=1091.659,-75.835,-51.103,174.880,16.078,152.463
C03380=1091.654,-76.085,-51.092,174.878,16.077,152.464
C03381=1091.648,-76.335,-51.081,174.877,16.077,152.464
C03382=1091.641,-76.585,-51.071,174.875,16.076,152.464
C03383=1091.635,-76.834,-51.060,174.874,16.075,152.464
C03384=1091.630,-77.084,-51.049,174.872,16.074,152.464
C03385=1091.624,-77.333,-51.038,174.870,16.073,152.464
C03386=1091.618,-77.583,-51.027,174.869,16.072,152.464
C03387=1091.612,-77.833,-51.016,174.867,16.071,152.465
C03388=1091.605,-78.082,-51.006,174.865,16.070,152.465
C03389=1091.600,-78.331,-50.995,174.864,16.070,152.465
C03390=1091.594,-78.582,-50.984,174.863,16.068,152.465
C03391=1091.588,-78.832,-50.974,174.861,16.068,152.465
C03392=1091.582,-79.081,-50.963,174.859,16.067,152.465
C03393=1091.576,-79.330,-50.952,174.857,16.066,152.466
C03394=1091.569,-79.581,-50.941,174.856,16.065,152.466
C03395=1091.564,-79.830,-50.930,174.854,16.064,152.466
C03396=1091.558,-80.080,-50.920,174.853,16.064,152.466
C03397=1091.552,-80.329,-50.910,174.851,16.062,152.466
C03398=1091.545,-80.603,-50.898,174.849,16.062,152.466
C03399=1091.538,-80.876,-50.886,174.848,16.061,152.467
C03400=1091.531,-81.150,-50.874,174.846,16.060,152.467
C03401=1091.526,-81.422,-50.862,174.844,16.059,152.467
C03402=1091.518,-81.672,-50.852,174.843,16.058,152.467
C03403=1091.513,-81.922,-50.842,174.841,16.057,152.467
C03404=1091.507,-82.172,-50.831,174.839,16.056,152.467
C03405=1091.501,-82.421,-50.821,174.837,16.055,152.468
C03406=1091.494,-82.671,-50.809,174.836,16.054,152.468
C03407=1091.488,-82.921,-50.800,174.834,16.054,152.468
C03408=1091.483,-83.171,-50.789,174.833,16.053,152.468
C03409=1091.477,-83.420,-50.778,174.831,16.052,152.468
C03410=1091.470,-83.670,-50.767,174.829,16.051,152.469
C03411=1091.464,-83.920,-50.757,174.828,16.050,152.469
C03412=1091.458,-84.169,-50.747,174.826,16.049,152.469
C03413=1091.452,-84.419,-50.736,174.825,16.049,152.469
C03414=1091.446,-84.668,-50.725,174.823,16.048,152.469
C03415=1091.440,-84.919,-50.715,174.822,16.047,152.469
C03416=1091.434,-85.168,-50.704,174.820,16.046,152.470
C03417=1091.428,-85.418,-50.693,174.818,16.045,152.470
C03418=1091.422,-85.667,-50.684,174.816,16.045,152.470
C03419=1091.416,-85.917,-50.673,174.815,16.044,152.470
C03420=1091.409,-86.167,-50.662,174.813,16.043,152.470
C03421=1091.404,-86.417,-50.652,174.812,16.042,152.470
C03422=1091.398,-86.666,-50.641,174.810,16.042,152.471
C03423=1091.391,-86.916,-50.631,174.808,16.040,152.471
C03424=1091.386,-87.166,-50.621,174.807,16.040,152.471
C03425=1091.379,-87.416,-50.610,174.806,16.039,152.471
C03426=1091.373,-87.665,-50.599,174.804,16.038,152.471
C03427=1091.367,-87.915,-50.590,174.802,16.037,152.471
C03428=1091.361,-88.164,-50.579,174.800,16.036,152.472
C03429=1091.356,-88.415,-50.569,174.799,16.036,152.472
C03430=1091.349,-88.664,-50.558,174.798,16.035,152.472
C03431=1091.343,-88.914,-50.547,174.796,16.034,152.472
C03432=1091.337,-89.164,-50.538,174.794,16.033,152.472
C03433=1091.331,-89.413,-50.527,174.792,16.033,152.473
C03434=1091.325,-89.663,-50.517,174.792,16.032,152.473
C03435=1091.319,-89.912,-50.506,174.790,16.031,152.473
C03436=1091.313,-90.162,-50.496,174.788,16.030,152.473
C03437=1091.307,-90.412,-50.486,174.786,16.030,152.473
C03438=1091.302,-90.661,-50.475,174.784,16.029,152.473
C03439=1091.295,-90.912,-50.465,174.783,16.028,152.474
C03440=1091.289,-91.161,-50.454,174.782,16.027,152.474
C03441=1091.283,-91.411,-50.445,174.780,16.027,152.474
C03442=1091.277,-91.660,-50.434,174.778,16.026,152.474
C03443=1091.271,-91.910,-50.424,174.776,16.025,152.474
C03444=1091.265,-92.160,-50.413,174.776,16.024,152.474
C03445=1091.259,-92.410,-50.404,174.774,16.024,152.475
C03446=1091.253,-92.659,-50.393,174.772,16.023,152.475
C03447=1091.247,-92.909,-50.383,174.770,16.022,152.475
C03448=1091.241,-93.159,-50.372,174.769,16.021,152.475
C03449=1091.235,-93.409,-50.362,174.767,16.021,152.475
C03450=1091.229,-93.658,-50.352,174.766,16.020,152.476
C03451=1091.223,-93.908,-50.342,174.764,16.019,152.476
C03452=1091.217,-94.158,-50.331,174.762,16.018,152.476
C03453=1091.211,-94.407,-50.322,174.761,16.018,152.476
C03454=1091.205,-94.657,-50.311,174.759,16.017,152.476
C03455=1091.199,-94.907,-50.301,174.758,16.016,152.476
C03456=1091.193,-95.156,-50.290,174.756,16.015,152.477
C03457=1091.187,-95.406,-50.281,174.754,16.014,152.477
C03458=1091.182,-95.656,-50.270,174.753,16.014,152.477
C03459=1091.175,-95.905,-50.260,174.751,16.013,152.477
C03460=1091.170,-96.155,-50.250,174.750,16.012,152.477
C03461=1091.163,-96.405,-50.240,174.748,16.011,152.477
C03462=1091.157,-96.680,-50.229,174.746,16.011,152.478
C03463=1091.150,-96.956,-50.217,174.745,16.010,152.478
C03464=1091.144,-97.232,-50.206,174.743,16.009,152.478
C03465=1091.137,-97.507,-50.195,174.741,16.009,152.478
C03466=1091.131,-97.757,-50.184,174.740,16.008,152.478
C03467=1091.125,-98.007,-50.175,174.738,16.007,152.479
C03468=1091.119,-98.256,-50.165,174.736,16.006,152.479
C03469=1091.113,-98.506,-50.154,174.735,16.006,152.479
C03470=1091.107,-98.756,-50.145,174.733,16.005,152.479
C03471=1091.101,-99.005,-50.135,174.731,16.004,152.480
C03472=1091.095,-99.255,-50.124,174.730,16.003,152.480
C03473=1091.089,-99.505,-50.115,174.729,16.003,152.480
C03474=1091.082,-99.755,-50.104,174.727,16.003,152.480
C03475=1091.075,-100.004,-50.095,174.725,16.001,152.480
C03476=1091.070,-100.255,-50.085,174.723,16.001,152.481
C03477=1091.063,-100.504,-50.074,174.722,16.001,152.481
C03478=1091.057,-100.753,-50.065,174.721,16.000,152.481
C03479=1091.052,-101.004,-50.055,174.719,15.999,152.481
C03480=1091.046,-101.253,-50.045,174.718,15.999,152.481
C03481=1091.039,-101.503,-50.035,174.716,15.998,152.481
C03482=1091.033,-101.752,-50.025,174.714,15.997,152.482
C03483=1091.028,-102.002,-50.015,174.712,15.996,152.482
C03484=1091.021,-102.252,-50.005,174.711,15.996,152.482
C03485=1091.015,-102.501,-49.995,174.709,15.995,152.482
C03486=1091.010,-102.752,-49.985,174.708,15.995,152.483
C03487=1091.003,-103.001,-49.975,174.706,15.993,152.483
C03488=1090.997,-103.251,-49.965,174.705,15.993,152.483
C03489=1090.991,-103.500,-49.955,174.703,15.993,152.483
C03490=1090.985,-103.750,-49.945,174.701,15.992,152.483
C03491=1090.979,-104.000,-49.936,174.700,15.992,152.484
C03492=1090.973,-104.249,-49.925,174.698,15.991,152.484
C03493=1090.966,-104.499,-49.916,174.696,15.990,152.484
C03494=1090.960,-104.749,-49.906,174.695,15.989,152.484
C03495=1090.955,-104.999,-49.896,174.694,15.989,152.484
C03496=1090.948,-105.248,-49.886,174.692,15.988,152.485
C03497=1090.942,-105.498,-49.876,174.690,15.987,152.485
C03498=1090.936,-105.748,-49.867,174.689,15.987,152.485
C03499=1090.931,-105.998,-49.857,174.687,15.987,152.485
C03500=1090.924,-106.248,-49.847,174.685,15.986,152.486
C03501=1090.918,-106.498,-49.837,174.684,15.985,152.486
C03502=1090.912,-106.747,-49.827,174.683,15.985,152.486
C03503=1090.906,-106.997,-49.818,174.681,15.984,152.486
C03504=1090.900,-107.247,-49.807,174.679,15.983,152.486
C03505=1090.894,-107.497,-49.798,174.678,15.983,152.486
C03506=1090.888,-107.746,-49.788,174.676,15.982,152.487
C03507=1090.882,-107.996,-49.779,174.674,15.982,152.487
C03508=1090.875,-108.245,-49.768,174.673,15.982,152.487
C03509=1090.869,-108.495,-49.759,174.671,15.980,152.487
C03510=1090.863,-108.745,-49.749,174.669,15.980,152.488
C03511=1090.857,-108.995,-49.740,174.668,15.980,152.488
C03512=1090.850,-109.244,-49.730,174.666,15.979,152.488
C03513=1090.845,-109.495,-49.720,174.665,15.978,152.488
C03514=1090.839,-109.744,-49.710,174.664,15.978,152.488
C03515=1090.833,-109.994,-49.701,174.662,15.977,152.489
C03516=1090.827,-110.243,-49.691,174.660,15.977,152.489
C03517=1090.821,-110.492,-49.681,174.658,15.976,152.489
C03518=1090.814,-110.742,-49.672,174.657,15.976,152.489
C03519=1090.808,-110.992,-49.662,174.655,15.975,152.490
C03520=1090.802,-111.242,-49.653,174.653,15.974,152.490
C03521=1090.796,-111.492,-49.643,174.652,15.974,152.490
C03522=1090.790,-111.741,-49.634,174.650,15.973,152.490
C03523=1090.784,-111.991,-49.624,174.648,15.973,152.491
C03524=1090.777,-112.241,-49.614,174.648,15.972,152.491
C03525=1090.771,-112.491,-49.605,174.646,15.972,152.491
C03526=1090.765,-112.759,-49.594,174.644,15.971,152.491
C03527=1090.759,-113.028,-49.584,174.643,15.971,152.491
C03528=1090.752,-113.297,-49.573,174.641,15.970,152.492
C03529=1090.745,-113.566,-49.563,174.639,15.970,152.492
C03530=1090.740,-113.815,-49.554,174.637,15.969,152.492
C03531=1090.734,-114.065,-49.545,174.636,15.969,152.492
C03532=1090.727,-114.315,-49.535,174.634,15.968,152.492
C03533=1090.721,-114.564,-49.526,174.632,15.967,152.493
C03534=1090.715,-114.814,-49.516,174.631,15.967,152.493
C03535=1090.709,-115.064,-49.506,174.629,15.966,152.493
C03536=1090.703,-115.314,-49.497,174.627,15.966,152.494
C03537=1090.697,-115.564,-49.487,174.626,15.966,152.494
C03538=1090.690,-115.813,-49.478,174.624,15.965,152.494
C03539=1090.684,-116.063,-49.468,174.623,15.964,152.494
C03540=1090.678,-116.313,-49.459,174.622,15.964,152.494
C03541=1090.673,-116.562,-49.449,174.620,15.963,152.495
C03542=1090.666,-116.812,-49.440,174.619,15.963,152.495
C03543=1090.659,-117.061,-49.431,174.617,15.963,152.495
C03544=1090.653,-117.311,-49.421,174.615,15.962,152.495
C03545=1090.647,-117.561,-49.412,174.614,15.962,152.496
C03546=1090.641,-117.811,-49.402,174.612,15.961,152.496
C03547=1090.635,-118.061,-49.393,174.610,15.961,152.496
C03548=1090.629,-118.310,-49.383,174.609,15.961,152.496
C03549=1090.622,-118.560,-49.373,174.607,15.960,152.497
C03550=1090.617,-118.809,-49.364,174.605,15.959,152.497
C03551=1090.611,-119.060,-49.355,174.604,15.959,152.497
C03552=1090.605,-119.310,-49.346,174.602,15.959,152.497
C03553=1090.599,-119.559,-49.336,174.601,15.958,152.497
C03554=1090.592,-119.809,-49.327,174.599,15.957,152.498
C03555=1090.586,-120.059,-49.318,174.597,15.957,152.498
C03556=1090.579,-120.308,-49.308,174.596,15.957,152.498
C03557=1090.573,-120.558,-49.299,174.594,15.956,152.498
C03558=1090.568,-120.807,-49.289,174.593,15.955,152.499
C03559=1090.562,-121.058,-49.280,174.591,15.955,152.499
C03560=1090.556,-121.308,-49.271,174.590,15.955,152.499
C03561=1090.549,-121.557,-49.261,174.588,15.955,152.499
C03562=1090.542,-121.807,-49.252,174.587,15.954,152.500
C03563=1090.536,-122.057,-49.243,174.585,15.953,152.500
C03564=1090.531,-122.306,-49.234,174.584,15.953,152.500
C03565=1090.525,-122.556,-49.225,174.582,15.953,152.500
C03566=1090.519,-122.806,-49.215,174.580,15.953,152.501
C03567=1090.513,-123.056,-49.206,174.579,15.952,152.501
C03568=1090.506,-123.305,-49.197,174.577,15.951,152.501
C03569=1090.499,-123.555,-49.187,174.576,15.951,152.501
C03570=1090.494,-123.805,-49.179,174.574,15.951,152.502
C03571=1090.488,-124.055,-49.169,174.573,15.951,152.502
C03572=1090.482,-124.304,-49.159,174.571,15.950,152.502
C03573=1090.476,-124.554,-49.150,174.569,15.949,152.502
C03574=1090.469,-124.804,-49.142,174.568,15.949,152.503
C03575=1090.463,-125.054,-49.132,174.566,15.949,152.503
C03576=1090.457,-125.303,-49.123,174.565,15.949,152.503
C03577=1090.451,-125.553,-49.113,174.563,15.948,152.503
C03578=1090.445,-125.803,-49.105,174.561,15.947,152.504
C03579=1090.438,-126.053,-49.095,174.560,15.947,152.504
C03580=1090.432,-126.303,-49.086,174.557,15.947,152.504
C03581=1090.426,-126.552,-49.076,174.556,15.947,152.505
C03582=1090.420,-126.802,-49.068,174.554,15.946,152.505
C03583=1090.414,-127.052,-49.059,174.553,15.946,152.505
C03584=1090.408,-127.301,-49.049,174.551,15.946,152.505
C03585=1090.401,-127.552,-49.041,174.550,15.945,152.506
C03586=1090.395,-127.810,-49.031,174.548,15.945,152.506
C03587=1090.389,-128.069,-49.021,174.547,15.944,152.506
C03588=1090.386,-128.327,-49.011,174.545,15.943,152.506
C03589=1090.392,-128.583,-48.999,174.545,15.940,152.506
C03590=1089.987,-128.604,-49.119,174.503,16.045,152.534
C03591=1089.981,-128.349,-49.132,174.503,16.049,152.535
C03592=1089.982,-128.090,-49.143,174.505,16.051,152.535
C03593=1089.989,-127.832,-49.152,174.506,16.051,152.535
C03594=1089.995,-127.573,-49.162,174.508,16.051,152.534
C03595=1090.002,-127.323,-49.171,174.510,16.052,152.534
C03596=1090.008,-127.074,-49.179,174.511,16.052,152.534
C03597=1090.014,-126.824,-49.189,174.513,16.053,152.534
C03598=1090.020,-126.574,-49.198,174.514,16.053,152.534
C03599=1090.027,-126.324,-49.207,174.516,16.053,152.533
C03600=1090.033,-126.074,-49.216,174.518,16.054,152.533
C03601=1090.038,-125.825,-49.225,174.519,16.054,152.533
C03602=1090.044,-125.575,-49.235,174.521,16.055,152.532
C03603=1090.051,-125.325,-49.243,174.522,16.055,152.532
C03604=1090.057,-125.075,-49.253,174.524,16.055,152.532
C03605=1090.063,-124.826,-49.262,174.525,16.055,152.532
C03606=1090.070,-124.576,-49.272,174.527,16.056,152.532
C03607=1090.076,-124.326,-49.280,174.528,16.057,152.531
C03608=1090.082,-124.077,-49.289,174.530,16.057,152.531
C03609=1090.088,-123.827,-49.299,174.532,16.057,152.531
C03610=1090.094,-123.577,-49.309,174.533,16.058,152.530
C03611=1090.100,-123.327,-49.318,174.535,16.058,152.530
C03612=1090.106,-123.077,-49.327,174.536,16.059,152.530
C03613=1090.112,-122.828,-49.336,174.538,16.059,152.530
C03614=1090.119,-122.578,-49.345,174.539,16.059,152.529
C03615=1090.125,-122.328,-49.355,174.541,16.060,152.529
C03616=1090.131,-122.079,-49.364,174.542,16.060,152.529
C03617=1090.137,-121.828,-49.373,174.544,16.061,152.529
C03618=1090.143,-121.578,-49.383,174.545,16.061,152.529
C03619=1090.149,-121.330,-49.391,174.547,16.061,152.528
C03620=1090.155,-121.080,-49.401,174.549,16.062,152.528
C03621=1090.162,-120.830,-49.410,174.550,16.062,152.528
C03622=1090.168,-120.580,-49.420,174.552,16.063,152.527
